  STRUCT
   FC2_RECV_1 : ARRAY  [0 .. 499 ] OF BYTE  := B#16#0;
  END_STRUCT ;
BEGIN
   FC2_RECV_1[0] := B#16#0;
   FC2_RECV_1[1] := B#16#0;
   FC2_RECV_1[2] := B#16#0;
   FC2_RECV_1[3] := B#16#0;
   FC2_RECV_1[4] := B#16#0;
   FC2_RECV_1[5] := B#16#0;
   FC2_RECV_1[6] := B#16#0;
   FC2_RECV_1[7] := B#16#0;
   FC2_RECV_1[8] := B#16#0;
   FC2_RECV_1[9] := B#16#0;
   FC2_RECV_1[10] := B#16#0;
   FC2_RECV_1[11] := B#16#0;
   FC2_RECV_1[12] := B#16#0;
   FC2_RECV_1[13] := B#16#0;
   FC2_RECV_1[14] := B#16#0;
   FC2_RECV_1[15] := B#16#0;
   FC2_RECV_1[16] := B#16#0;
   FC2_RECV_1[17] := B#16#0;
   FC2_RECV_1[18] := B#16#0;
   FC2_RECV_1[19] := B#16#0;
   FC2_RECV_1[20] := B#16#0;
   FC2_RECV_1[21] := B#16#0;
   FC2_RECV_1[22] := B#16#0;
   FC2_RECV_1[23] := B#16#0;
   FC2_RECV_1[24] := B#16#0;
   FC2_RECV_1[25] := B#16#0;
   FC2_RECV_1[26] := B#16#0;
   FC2_RECV_1[27] := B#16#0;
   FC2_RECV_1[28] := B#16#0;
   FC2_RECV_1[29] := B#16#0;
   FC2_RECV_1[30] := B#16#0;
   FC2_RECV_1[31] := B#16#0;
   FC2_RECV_1[32] := B#16#0;
   FC2_RECV_1[33] := B#16#0;
   FC2_RECV_1[34] := B#16#0;
   FC2_RECV_1[35] := B#16#0;
   FC2_RECV_1[36] := B#16#0;
   FC2_RECV_1[37] := B#16#0;
   FC2_RECV_1[38] := B#16#0;
   FC2_RECV_1[39] := B#16#0;
   FC2_RECV_1[40] := B#16#0;
   FC2_RECV_1[41] := B#16#0;
   FC2_RECV_1[42] := B#16#0;
   FC2_RECV_1[43] := B#16#0;
   FC2_RECV_1[44] := B#16#0;
   FC2_RECV_1[45] := B#16#0;
   FC2_RECV_1[46] := B#16#0;
   FC2_RECV_1[47] := B#16#0;
   FC2_RECV_1[48] := B#16#0;
   FC2_RECV_1[49] := B#16#0;
   FC2_RECV_1[50] := B#16#0;
   FC2_RECV_1[51] := B#16#0;
   FC2_RECV_1[52] := B#16#0;
   FC2_RECV_1[53] := B#16#0;
   FC2_RECV_1[54] := B#16#0;
   FC2_RECV_1[55] := B#16#0;
   FC2_RECV_1[56] := B#16#0;
   FC2_RECV_1[57] := B#16#0;
   FC2_RECV_1[58] := B#16#0;
   FC2_RECV_1[59] := B#16#0;
   FC2_RECV_1[60] := B#16#0;
   FC2_RECV_1[61] := B#16#0;
   FC2_RECV_1[62] := B#16#0;
   FC2_RECV_1[63] := B#16#0;
   FC2_RECV_1[64] := B#16#0;
   FC2_RECV_1[65] := B#16#0;
   FC2_RECV_1[66] := B#16#0;
   FC2_RECV_1[67] := B#16#0;
   FC2_RECV_1[68] := B#16#0;
   FC2_RECV_1[69] := B#16#0;
   FC2_RECV_1[70] := B#16#0;
   FC2_RECV_1[71] := B#16#0;
   FC2_RECV_1[72] := B#16#0;
   FC2_RECV_1[73] := B#16#0;
   FC2_RECV_1[74] := B#16#0;
   FC2_RECV_1[75] := B#16#0;
   FC2_RECV_1[76] := B#16#0;
   FC2_RECV_1[77] := B#16#0;
   FC2_RECV_1[78] := B#16#0;
   FC2_RECV_1[79] := B#16#0;
   FC2_RECV_1[80] := B#16#0;
   FC2_RECV_1[81] := B#16#0;
   FC2_RECV_1[82] := B#16#0;
   FC2_RECV_1[83] := B#16#0;
   FC2_RECV_1[84] := B#16#0;
   FC2_RECV_1[85] := B#16#0;
   FC2_RECV_1[86] := B#16#0;
   FC2_RECV_1[87] := B#16#0;
   FC2_RECV_1[88] := B#16#0;
   FC2_RECV_1[89] := B#16#0;
   FC2_RECV_1[90] := B#16#0;
   FC2_RECV_1[91] := B#16#0;
   FC2_RECV_1[92] := B#16#0;
   FC2_RECV_1[93] := B#16#0;
   FC2_RECV_1[94] := B#16#0;
   FC2_RECV_1[95] := B#16#0;
   FC2_RECV_1[96] := B#16#0;
   FC2_RECV_1[97] := B#16#0;
   FC2_RECV_1[98] := B#16#0;
   FC2_RECV_1[99] := B#16#0;
   FC2_RECV_1[100] := B#16#0;
   FC2_RECV_1[101] := B#16#0;
   FC2_RECV_1[102] := B#16#0;
   FC2_RECV_1[103] := B#16#0;
   FC2_RECV_1[104] := B#16#0;
   FC2_RECV_1[105] := B#16#0;
   FC2_RECV_1[106] := B#16#0;
   FC2_RECV_1[107] := B#16#0;
   FC2_RECV_1[108] := B#16#0;
   FC2_RECV_1[109] := B#16#0;
   FC2_RECV_1[110] := B#16#0;
   FC2_RECV_1[111] := B#16#0;
   FC2_RECV_1[112] := B#16#0;
   FC2_RECV_1[113] := B#16#0;
   FC2_RECV_1[114] := B#16#0;
   FC2_RECV_1[115] := B#16#0;
   FC2_RECV_1[116] := B#16#0;
   FC2_RECV_1[117] := B#16#0;
   FC2_RECV_1[118] := B#16#0;
   FC2_RECV_1[119] := B#16#0;
   FC2_RECV_1[120] := B#16#0;
   FC2_RECV_1[121] := B#16#0;
   FC2_RECV_1[122] := B#16#0;
   FC2_RECV_1[123] := B#16#0;
   FC2_RECV_1[124] := B#16#0;
   FC2_RECV_1[125] := B#16#0;
   FC2_RECV_1[126] := B#16#0;
   FC2_RECV_1[127] := B#16#0;
   FC2_RECV_1[128] := B#16#0;
   FC2_RECV_1[129] := B#16#0;
   FC2_RECV_1[130] := B#16#0;
   FC2_RECV_1[131] := B#16#0;
   FC2_RECV_1[132] := B#16#0;
   FC2_RECV_1[133] := B#16#0;
   FC2_RECV_1[134] := B#16#0;
   FC2_RECV_1[135] := B#16#0;
   FC2_RECV_1[136] := B#16#0;
   FC2_RECV_1[137] := B#16#0;
   FC2_RECV_1[138] := B#16#0;
   FC2_RECV_1[139] := B#16#0;
   FC2_RECV_1[140] := B#16#0;
   FC2_RECV_1[141] := B#16#0;
   FC2_RECV_1[142] := B#16#0;
   FC2_RECV_1[143] := B#16#0;
   FC2_RECV_1[144] := B#16#0;
   FC2_RECV_1[145] := B#16#0;
   FC2_RECV_1[146] := B#16#0;
   FC2_RECV_1[147] := B#16#0;
   FC2_RECV_1[148] := B#16#0;
   FC2_RECV_1[149] := B#16#0;
   FC2_RECV_1[150] := B#16#0;
   FC2_RECV_1[151] := B#16#0;
   FC2_RECV_1[152] := B#16#0;
   FC2_RECV_1[153] := B#16#0;
   FC2_RECV_1[154] := B#16#0;
   FC2_RECV_1[155] := B#16#0;
   FC2_RECV_1[156] := B#16#0;
   FC2_RECV_1[157] := B#16#0;
   FC2_RECV_1[158] := B#16#0;
   FC2_RECV_1[159] := B#16#0;
   FC2_RECV_1[160] := B#16#0;
   FC2_RECV_1[161] := B#16#0;
   FC2_RECV_1[162] := B#16#0;
   FC2_RECV_1[163] := B#16#0;
   FC2_RECV_1[164] := B#16#0;
   FC2_RECV_1[165] := B#16#0;
   FC2_RECV_1[166] := B#16#0;
   FC2_RECV_1[167] := B#16#0;
   FC2_RECV_1[168] := B#16#0;
   FC2_RECV_1[169] := B#16#0;
   FC2_RECV_1[170] := B#16#0;
   FC2_RECV_1[171] := B#16#0;
   FC2_RECV_1[172] := B#16#0;
   FC2_RECV_1[173] := B#16#0;
   FC2_RECV_1[174] := B#16#0;
   FC2_RECV_1[175] := B#16#0;
   FC2_RECV_1[176] := B#16#0;
   FC2_RECV_1[177] := B#16#0;
   FC2_RECV_1[178] := B#16#0;
   FC2_RECV_1[179] := B#16#0;
   FC2_RECV_1[180] := B#16#0;
   FC2_RECV_1[181] := B#16#0;
   FC2_RECV_1[182] := B#16#0;
   FC2_RECV_1[183] := B#16#0;
   FC2_RECV_1[184] := B#16#0;
   FC2_RECV_1[185] := B#16#0;
   FC2_RECV_1[186] := B#16#0;
   FC2_RECV_1[187] := B#16#0;
   FC2_RECV_1[188] := B#16#0;
   FC2_RECV_1[189] := B#16#0;
   FC2_RECV_1[190] := B#16#0;
   FC2_RECV_1[191] := B#16#0;
   FC2_RECV_1[192] := B#16#0;
   FC2_RECV_1[193] := B#16#0;
   FC2_RECV_1[194] := B#16#0;
   FC2_RECV_1[195] := B#16#0;
   FC2_RECV_1[196] := B#16#0;
   FC2_RECV_1[197] := B#16#0;
   FC2_RECV_1[198] := B#16#0;
   FC2_RECV_1[199] := B#16#0;
   FC2_RECV_1[200] := B#16#0;
   FC2_RECV_1[201] := B#16#0;
   FC2_RECV_1[202] := B#16#0;
   FC2_RECV_1[203] := B#16#0;
   FC2_RECV_1[204] := B#16#0;
   FC2_RECV_1[205] := B#16#0;
   FC2_RECV_1[206] := B#16#0;
   FC2_RECV_1[207] := B#16#0;
   FC2_RECV_1[208] := B#16#0;
   FC2_RECV_1[209] := B#16#0;
   FC2_RECV_1[210] := B#16#0;
   FC2_RECV_1[211] := B#16#0;
   FC2_RECV_1[212] := B#16#0;
   FC2_RECV_1[213] := B#16#0;
   FC2_RECV_1[214] := B#16#0;
   FC2_RECV_1[215] := B#16#0;
   FC2_RECV_1[216] := B#16#0;
   FC2_RECV_1[217] := B#16#0;
   FC2_RECV_1[218] := B#16#0;
   FC2_RECV_1[219] := B#16#0;
   FC2_RECV_1[220] := B#16#0;
   FC2_RECV_1[221] := B#16#0;
   FC2_RECV_1[222] := B#16#0;
   FC2_RECV_1[223] := B#16#0;
   FC2_RECV_1[224] := B#16#0;
   FC2_RECV_1[225] := B#16#0;
   FC2_RECV_1[226] := B#16#0;
   FC2_RECV_1[227] := B#16#0;
   FC2_RECV_1[228] := B#16#0;
   FC2_RECV_1[229] := B#16#0;
   FC2_RECV_1[230] := B#16#0;
   FC2_RECV_1[231] := B#16#0;
   FC2_RECV_1[232] := B#16#0;
   FC2_RECV_1[233] := B#16#0;
   FC2_RECV_1[234] := B#16#0;
   FC2_RECV_1[235] := B#16#0;
   FC2_RECV_1[236] := B#16#0;
   FC2_RECV_1[237] := B#16#0;
   FC2_RECV_1[238] := B#16#0;
   FC2_RECV_1[239] := B#16#0;
   FC2_RECV_1[240] := B#16#0;
   FC2_RECV_1[241] := B#16#0;
   FC2_RECV_1[242] := B#16#0;
   FC2_RECV_1[243] := B#16#0;
   FC2_RECV_1[244] := B#16#0;
   FC2_RECV_1[245] := B#16#0;
   FC2_RECV_1[246] := B#16#0;
   FC2_RECV_1[247] := B#16#0;
   FC2_RECV_1[248] := B#16#0;
   FC2_RECV_1[249] := B#16#0;
   FC2_RECV_1[250] := B#16#0;
   FC2_RECV_1[251] := B#16#0;
   FC2_RECV_1[252] := B#16#0;
   FC2_RECV_1[253] := B#16#0;
   FC2_RECV_1[254] := B#16#0;
   FC2_RECV_1[255] := B#16#0;
   FC2_RECV_1[256] := B#16#0;
   FC2_RECV_1[257] := B#16#0;
   FC2_RECV_1[258] := B#16#0;
   FC2_RECV_1[259] := B#16#0;
   FC2_RECV_1[260] := B#16#0;
   FC2_RECV_1[261] := B#16#0;
   FC2_RECV_1[262] := B#16#0;
   FC2_RECV_1[263] := B#16#0;
   FC2_RECV_1[264] := B#16#0;
   FC2_RECV_1[265] := B#16#0;
   FC2_RECV_1[266] := B#16#0;
   FC2_RECV_1[267] := B#16#0;
   FC2_RECV_1[268] := B#16#0;
   FC2_RECV_1[269] := B#16#0;
   FC2_RECV_1[270] := B#16#0;
   FC2_RECV_1[271] := B#16#0;
   FC2_RECV_1[272] := B#16#0;
   FC2_RECV_1[273] := B#16#0;
   FC2_RECV_1[274] := B#16#0;
   FC2_RECV_1[275] := B#16#0;
   FC2_RECV_1[276] := B#16#0;
   FC2_RECV_1[277] := B#16#0;
   FC2_RECV_1[278] := B#16#0;
   FC2_RECV_1[279] := B#16#0;
   FC2_RECV_1[280] := B#16#0;
   FC2_RECV_1[281] := B#16#0;
   FC2_RECV_1[282] := B#16#0;
   FC2_RECV_1[283] := B#16#0;
   FC2_RECV_1[284] := B#16#0;
   FC2_RECV_1[285] := B#16#0;
   FC2_RECV_1[286] := B#16#0;
   FC2_RECV_1[287] := B#16#0;
   FC2_RECV_1[288] := B#16#0;
   FC2_RECV_1[289] := B#16#0;
   FC2_RECV_1[290] := B#16#0;
   FC2_RECV_1[291] := B#16#0;
   FC2_RECV_1[292] := B#16#0;
   FC2_RECV_1[293] := B#16#0;
   FC2_RECV_1[294] := B#16#0;
   FC2_RECV_1[295] := B#16#0;
   FC2_RECV_1[296] := B#16#0;
   FC2_RECV_1[297] := B#16#0;
   FC2_RECV_1[298] := B#16#0;
   FC2_RECV_1[299] := B#16#0;
   FC2_RECV_1[300] := B#16#0;
   FC2_RECV_1[301] := B#16#0;
   FC2_RECV_1[302] := B#16#0;
   FC2_RECV_1[303] := B#16#0;
   FC2_RECV_1[304] := B#16#0;
   FC2_RECV_1[305] := B#16#0;
   FC2_RECV_1[306] := B#16#0;
   FC2_RECV_1[307] := B#16#0;
   FC2_RECV_1[308] := B#16#0;
   FC2_RECV_1[309] := B#16#0;
   FC2_RECV_1[310] := B#16#0;
   FC2_RECV_1[311] := B#16#0;
   FC2_RECV_1[312] := B#16#0;
   FC2_RECV_1[313] := B#16#0;
   FC2_RECV_1[314] := B#16#0;
   FC2_RECV_1[315] := B#16#0;
   FC2_RECV_1[316] := B#16#0;
   FC2_RECV_1[317] := B#16#0;
   FC2_RECV_1[318] := B#16#0;
   FC2_RECV_1[319] := B#16#0;
   FC2_RECV_1[320] := B#16#0;
   FC2_RECV_1[321] := B#16#0;
   FC2_RECV_1[322] := B#16#0;
   FC2_RECV_1[323] := B#16#0;
   FC2_RECV_1[324] := B#16#0;
   FC2_RECV_1[325] := B#16#0;
   FC2_RECV_1[326] := B#16#0;
   FC2_RECV_1[327] := B#16#0;
   FC2_RECV_1[328] := B#16#0;
   FC2_RECV_1[329] := B#16#0;
   FC2_RECV_1[330] := B#16#0;
   FC2_RECV_1[331] := B#16#0;
   FC2_RECV_1[332] := B#16#0;
   FC2_RECV_1[333] := B#16#0;
   FC2_RECV_1[334] := B#16#0;
   FC2_RECV_1[335] := B#16#0;
   FC2_RECV_1[336] := B#16#0;
   FC2_RECV_1[337] := B#16#0;
   FC2_RECV_1[338] := B#16#0;
   FC2_RECV_1[339] := B#16#0;
   FC2_RECV_1[340] := B#16#0;
   FC2_RECV_1[341] := B#16#0;
   FC2_RECV_1[342] := B#16#0;
   FC2_RECV_1[343] := B#16#0;
   FC2_RECV_1[344] := B#16#0;
   FC2_RECV_1[345] := B#16#0;
   FC2_RECV_1[346] := B#16#0;
   FC2_RECV_1[347] := B#16#0;
   FC2_RECV_1[348] := B#16#0;
   FC2_RECV_1[349] := B#16#0;
   FC2_RECV_1[350] := B#16#0;
   FC2_RECV_1[351] := B#16#0;
   FC2_RECV_1[352] := B#16#0;
   FC2_RECV_1[353] := B#16#0;
   FC2_RECV_1[354] := B#16#0;
   FC2_RECV_1[355] := B#16#0;
   FC2_RECV_1[356] := B#16#0;
   FC2_RECV_1[357] := B#16#0;
   FC2_RECV_1[358] := B#16#0;
   FC2_RECV_1[359] := B#16#0;
   FC2_RECV_1[360] := B#16#0;
   FC2_RECV_1[361] := B#16#0;
   FC2_RECV_1[362] := B#16#0;
   FC2_RECV_1[363] := B#16#0;
   FC2_RECV_1[364] := B#16#0;
   FC2_RECV_1[365] := B#16#0;
   FC2_RECV_1[366] := B#16#0;
   FC2_RECV_1[367] := B#16#0;
   FC2_RECV_1[368] := B#16#0;
   FC2_RECV_1[369] := B#16#0;
   FC2_RECV_1[370] := B#16#0;
   FC2_RECV_1[371] := B#16#0;
   FC2_RECV_1[372] := B#16#0;
   FC2_RECV_1[373] := B#16#0;
   FC2_RECV_1[374] := B#16#0;
   FC2_RECV_1[375] := B#16#0;
   FC2_RECV_1[376] := B#16#0;
   FC2_RECV_1[377] := B#16#0;
   FC2_RECV_1[378] := B#16#0;
   FC2_RECV_1[379] := B#16#0;
   FC2_RECV_1[380] := B#16#0;
   FC2_RECV_1[381] := B#16#0;
   FC2_RECV_1[382] := B#16#0;
   FC2_RECV_1[383] := B#16#0;
   FC2_RECV_1[384] := B#16#0;
   FC2_RECV_1[385] := B#16#0;
   FC2_RECV_1[386] := B#16#0;
   FC2_RECV_1[387] := B#16#0;
   FC2_RECV_1[388] := B#16#0;
   FC2_RECV_1[389] := B#16#0;
   FC2_RECV_1[390] := B#16#0;
   FC2_RECV_1[391] := B#16#0;
   FC2_RECV_1[392] := B#16#0;
   FC2_RECV_1[393] := B#16#0;
   FC2_RECV_1[394] := B#16#0;
   FC2_RECV_1[395] := B#16#0;
   FC2_RECV_1[396] := B#16#0;
   FC2_RECV_1[397] := B#16#0;
   FC2_RECV_1[398] := B#16#0;
   FC2_RECV_1[399] := B#16#0;
   FC2_RECV_1[400] := B#16#0;
   FC2_RECV_1[401] := B#16#0;
   FC2_RECV_1[402] := B#16#0;
   FC2_RECV_1[403] := B#16#0;
   FC2_RECV_1[404] := B#16#0;
   FC2_RECV_1[405] := B#16#0;
   FC2_RECV_1[406] := B#16#0;
   FC2_RECV_1[407] := B#16#0;
   FC2_RECV_1[408] := B#16#0;
   FC2_RECV_1[409] := B#16#0;
   FC2_RECV_1[410] := B#16#0;
   FC2_RECV_1[411] := B#16#0;
   FC2_RECV_1[412] := B#16#0;
   FC2_RECV_1[413] := B#16#0;
   FC2_RECV_1[414] := B#16#0;
   FC2_RECV_1[415] := B#16#0;
   FC2_RECV_1[416] := B#16#0;
   FC2_RECV_1[417] := B#16#0;
   FC2_RECV_1[418] := B#16#0;
   FC2_RECV_1[419] := B#16#0;
   FC2_RECV_1[420] := B#16#0;
   FC2_RECV_1[421] := B#16#0;
   FC2_RECV_1[422] := B#16#0;
   FC2_RECV_1[423] := B#16#0;
   FC2_RECV_1[424] := B#16#0;
   FC2_RECV_1[425] := B#16#0;
   FC2_RECV_1[426] := B#16#0;
   FC2_RECV_1[427] := B#16#0;
   FC2_RECV_1[428] := B#16#0;
   FC2_RECV_1[429] := B#16#0;
   FC2_RECV_1[430] := B#16#0;
   FC2_RECV_1[431] := B#16#0;
   FC2_RECV_1[432] := B#16#0;
   FC2_RECV_1[433] := B#16#0;
   FC2_RECV_1[434] := B#16#0;
   FC2_RECV_1[435] := B#16#0;
   FC2_RECV_1[436] := B#16#0;
   FC2_RECV_1[437] := B#16#0;
   FC2_RECV_1[438] := B#16#0;
   FC2_RECV_1[439] := B#16#0;
   FC2_RECV_1[440] := B#16#0;
   FC2_RECV_1[441] := B#16#0;
   FC2_RECV_1[442] := B#16#0;
   FC2_RECV_1[443] := B#16#0;
   FC2_RECV_1[444] := B#16#0;
   FC2_RECV_1[445] := B#16#0;
   FC2_RECV_1[446] := B#16#0;
   FC2_RECV_1[447] := B#16#0;
   FC2_RECV_1[448] := B#16#0;
   FC2_RECV_1[449] := B#16#0;
   FC2_RECV_1[450] := B#16#0;
   FC2_RECV_1[451] := B#16#0;
   FC2_RECV_1[452] := B#16#0;
   FC2_RECV_1[453] := B#16#0;
   FC2_RECV_1[454] := B#16#0;
   FC2_RECV_1[455] := B#16#0;
   FC2_RECV_1[456] := B#16#0;
   FC2_RECV_1[457] := B#16#0;
   FC2_RECV_1[458] := B#16#0;
   FC2_RECV_1[459] := B#16#0;
   FC2_RECV_1[460] := B#16#0;
   FC2_RECV_1[461] := B#16#0;
   FC2_RECV_1[462] := B#16#0;
   FC2_RECV_1[463] := B#16#0;
   FC2_RECV_1[464] := B#16#0;
   FC2_RECV_1[465] := B#16#0;
   FC2_RECV_1[466] := B#16#0;
   FC2_RECV_1[467] := B#16#0;
   FC2_RECV_1[468] := B#16#0;
   FC2_RECV_1[469] := B#16#0;
   FC2_RECV_1[470] := B#16#0;
   FC2_RECV_1[471] := B#16#0;
   FC2_RECV_1[472] := B#16#0;
   FC2_RECV_1[473] := B#16#0;
   FC2_RECV_1[474] := B#16#0;
   FC2_RECV_1[475] := B#16#0;
   FC2_RECV_1[476] := B#16#0;
   FC2_RECV_1[477] := B#16#0;
   FC2_RECV_1[478] := B#16#0;
   FC2_RECV_1[479] := B#16#0;
   FC2_RECV_1[480] := B#16#0;
   FC2_RECV_1[481] := B#16#0;
   FC2_RECV_1[482] := B#16#0;
   FC2_RECV_1[483] := B#16#0;
   FC2_RECV_1[484] := B#16#0;
   FC2_RECV_1[485] := B#16#0;
   FC2_RECV_1[486] := B#16#0;
   FC2_RECV_1[487] := B#16#0;
   FC2_RECV_1[488] := B#16#0;
   FC2_RECV_1[489] := B#16#0;
   FC2_RECV_1[490] := B#16#0;
   FC2_RECV_1[491] := B#16#0;
   FC2_RECV_1[492] := B#16#0;
   FC2_RECV_1[493] := B#16#0;
   FC2_RECV_1[494] := B#16#0;
   FC2_RECV_1[495] := B#16#0;
   FC2_RECV_1[496] := B#16#0;
   FC2_RECV_1[497] := B#16#0;
   FC2_RECV_1[498] := B#16#0;
   FC2_RECV_1[499] := B#16#0;
END_DATA_BLOCK

DATA_BLOCK DB 98
VERSION : 0.1


  STRUCT
   STAT0 : ARRAY  [0 .. 25 ] OF DWORD ;
  END_STRUCT ;
BEGIN
   STAT0[0] := DW#16#0;
   STAT0[1] := DW#16#0;
   STAT0[2] := DW#16#0;
   STAT0[3] := DW#16#0;
   STAT0[4] := DW#16#0;
   STAT0[5] := DW#16#0;
   STAT0[6] := DW#16#0;
   STAT0[7] := DW#16#0;
   STAT0[8] := DW#16#0;
   STAT0[9] := DW#16#0;
   STAT0[10] := DW#16#10000;
   STAT0[11] := DW#16#0;
   STAT0[12] := DW#16#0;
   STAT0[13] := DW#16#0;
   STAT0[14] := DW#16#0;
   STAT0[15] := DW#16#0;
   STAT0[16] := DW#16#0;
   STAT0[17] := DW#16#0;
   STAT0[18] := DW#16#0;
   STAT0[19] := DW#16#0;
   STAT0[20] := DW#16#0;
   STAT0[21] := DW#16#0;
   STAT0[22] := DW#16#0;
   STAT0[23] := DW#16#0;
   STAT0[24] := DW#16#0;
   STAT0[25] := DW#16#0;
END_DATA_BLOCK

DATA_BLOCK DB 99
VERSION : 0.1


  STRUCT
   STAT0 : WORD ;
   STAT1 : WORD ;
   STAT2 : WORD ;
   STAT3 : WORD ;
   STAT4 : WORD ;
   STAT5 : WORD ;
   STAT6 : WORD ;
   STAT7 : WORD ;
   STAT8 : WORD ;
   STAT9 : WORD ;
   STAT10 : WORD ;
   STAT11 : WORD ;
   STAT12 : WORD ;
   STAT13 : WORD ;
   STAT14 : WORD ;
   STAT15 : WORD ;
   STAT16 : WORD ;
   STAT17 : WORD ;
   STAT18 : WORD ;
   STAT19 : WORD ;
   STAT20 : WORD ;
   STAT21 : WORD ;
   STAT22 : WORD ;
   STAT23 : WORD ;
   STAT24 : WORD ;
   STAT25 : WORD ;
   STAT26 : WORD ;
   STAT27 : WORD ;
   STAT28 : WORD ;
   STAT29 : WORD ;
   STAT30 : WORD ;
   STAT31 : WORD ;
   STAT32 : WORD ;
   STAT33 : WORD ;
   STAT34 : WORD ;
   STAT35 : WORD ;
   STAT36 : WORD ;
   STAT37 : WORD ;
   STAT38 : WORD ;
   STAT39 : WORD ;
   STAT40 : WORD ;
   STAT41 : WORD ;
   STAT42 : WORD ;
   STAT43 : WORD ;
   STAT44 : WORD ;
   STAT45 : WORD ;
   STAT46 : WORD ;
   STAT47 : WORD ;
   STAT48 : WORD ;
   STAT49 : WORD ;
   STAT50 : WORD ;
   STAT51 : WORD ;
   STAT52 : WORD ;
   STAT53 : WORD ;
   STAT54 : WORD ;
   STAT55 : WORD ;
   STAT56 : WORD ;
   STAT57 : WORD ;
   STAT58 : WORD ;
   STAT59 : WORD ;
   STAT60 : WORD ;
   STAT61 : WORD ;
   STAT62 : WORD ;
   STAT63 : WORD ;
  END_STRUCT ;
BEGIN
   STAT0 := W#16#4101;
   STAT1 := W#16#9000;
   STAT2 := W#16#800;
   STAT3 := W#16#0;
   STAT4 := W#16#4102;
   STAT5 := W#16#9000;
   STAT6 := W#16#800;
   STAT7 := W#16#0;
   STAT8 := W#16#4201;
   STAT9 := W#16#5000;
   STAT10 := W#16#800;
   STAT11 := W#16#0;
   STAT12 := W#16#4102;
   STAT13 := W#16#9000;
   STAT14 := W#16#800;
   STAT15 := W#16#0;
   STAT16 := W#16#4101;
   STAT17 := W#16#9000;
   STAT18 := W#16#800;
   STAT19 := W#16#0;
   STAT20 := W#16#4101;
   STAT21 := W#16#9000;
   STAT22 := W#16#800;
   STAT23 := W#16#0;
   STAT24 := W#16#0;
   STAT25 := W#16#0;
   STAT26 := W#16#0;
   STAT27 := W#16#0;
   STAT28 := W#16#0;
   STAT29 := W#16#0;
   STAT30 := W#16#0;
   STAT31 := W#16#0;
   STAT32 := W#16#0;
   STAT33 := W#16#0;
   STAT34 := W#16#0;
   STAT35 := W#16#0;
   STAT36 := W#16#0;
   STAT37 := W#16#0;
   STAT38 := W#16#0;
   STAT39 := W#16#0;
   STAT40 := W#16#0;
   STAT41 := W#16#0;
   STAT42 := W#16#0;
   STAT43 := W#16#0;
   STAT44 := W#16#0;
   STAT45 := W#16#4102;
   STAT46 := W#16#9000;
   STAT47 := W#16#4201;
   STAT48 := W#16#5000;
   STAT49 := W#16#4102;
   STAT50 := W#16#9000;
   STAT51 := W#16#4201;
   STAT52 := W#16#5000;
   STAT53 := W#16#4101;
   STAT54 := W#16#9000;
   STAT55 := W#16#800;
   STAT56 := W#16#0;
   STAT57 := W#16#0;
   STAT58 := W#16#0;
   STAT59 := W#16#0;
   STAT60 := W#16#0;
   STAT61 := W#16#0;
   STAT62 := W#16#0;
   STAT63 := W#16#0;
END_DATA_BLOCK

DATA_BLOCK DB 100
VERSION : 0.1


  STRUCT
   STAT0 : WORD ;
   STAT1 : WORD ;
   STAT2 : WORD ;
   STAT3 : WORD ;
   STAT4 : WORD ;
   STAT5 : WORD ;
   STAT6 : WORD ;
   STAT7 : WORD ;
   STAT8 : WORD ;
   STAT9 : WORD ;
   STAT10 : WORD ;
   STAT11 : WORD ;
   STAT12 : WORD ;
   STAT13 : WORD ;
   STAT14 : WORD ;
   STAT15 : WORD ;
   STAT16 : WORD ;
   STAT17 : WORD ;
   STAT18 : WORD ;
   STAT19 : WORD ;
   STAT20 : WORD ;
   STAT21 : WORD ;
   STAT22 : WORD ;
   STAT23 : WORD ;
   STAT24 : WORD ;
   STAT25 : WORD ;
   STAT26 : WORD ;
   STAT27 : WORD ;
   STAT28 : WORD ;
   STAT29 : WORD ;
   STAT30 : WORD ;
   STAT31 : WORD ;
   STAT32 : WORD ;
   STAT33 : WORD ;
   STAT34 : WORD ;
   STAT35 : WORD ;
   STAT36 : WORD ;
   STAT37 : WORD ;
   STAT38 : WORD ;
   STAT39 : WORD ;
   STAT40 : WORD ;
   STAT41 : WORD ;
   STAT42 : WORD ;
   STAT43 : WORD ;
   STAT44 : WORD ;
   STAT45 : WORD ;
   STAT46 : WORD ;
   STAT47 : WORD ;
   STAT48 : WORD ;
   STAT49 : WORD ;
   STAT50 : WORD ;
   STAT51 : WORD ;
   STAT52 : WORD ;
   STAT53 : WORD ;
   STAT54 : WORD ;
   STAT55 : WORD ;
   STAT56 : WORD ;
   STAT57 : WORD ;
   STAT58 : WORD ;
   STAT59 : WORD ;
   STAT60 : WORD ;
   STAT61 : WORD ;
   STAT62 : WORD ;
   STAT63 : WORD ;
   STAT64 : WORD ;
   STAT65 : WORD ;
   STAT66 : WORD ;
   STAT67 : WORD ;
   STAT68 : WORD ;
   STAT69 : WORD ;
   STAT70 : WORD ;
   STAT71 : WORD ;
   STAT72 : WORD ;
   STAT73 : WORD ;
   STAT74 : WORD ;
   STAT75 : WORD ;
   STAT76 : WORD ;
   STAT77 : WORD ;
   STAT78 : WORD ;
   STAT79 : WORD ;
  END_STRUCT ;
BEGIN
   STAT0 := W#16#0;
   STAT1 := W#16#0;
   STAT2 := W#16#0;
   STAT3 := W#16#0;
   STAT4 := W#16#0;
   STAT5 := W#16#0;
   STAT6 := W#16#0;
   STAT7 := W#16#0;
   STAT8 := W#16#4201;
   STAT9 := W#16#5000;
   STAT10 := W#16#800;
   STAT11 := W#16#0;
   STAT12 := W#16#4102;
   STAT13 := W#16#9000;
   STAT14 := W#16#800;
   STAT15 := W#16#0;
   STAT16 := W#16#4101;
   STAT17 := W#16#9000;
   STAT18 := W#16#800;
   STAT19 := W#16#0;
   STAT20 := W#16#4201;
   STAT21 := W#16#5000;
   STAT22 := W#16#800;
   STAT23 := W#16#0;
   STAT24 := W#16#4102;
   STAT25 := W#16#9000;
   STAT26 := W#16#800;
   STAT27 := W#16#0;
   STAT28 := W#16#4101;
   STAT29 := W#16#9000;
   STAT30 := W#16#800;
   STAT31 := W#16#0;
   STAT32 := W#16#4102;
   STAT33 := W#16#A000;
   STAT34 := W#16#1000;
   STAT35 := W#16#0;
   STAT36 := W#16#4201;
   STAT37 := W#16#5000;
   STAT38 := W#16#800;
   STAT39 := W#16#0;
   STAT40 := W#16#4101;
   STAT41 := W#16#9000;
   STAT42 := W#16#800;
   STAT43 := W#16#0;
   STAT44 := W#16#0;
   STAT45 := W#16#0;
   STAT46 := W#16#0;
   STAT47 := W#16#0;
   STAT48 := W#16#0;
   STAT49 := W#16#0;
   STAT50 := W#16#0;
   STAT51 := W#16#0;
   STAT52 := W#16#0;
   STAT53 := W#16#0;
   STAT54 := W#16#0;
   STAT55 := W#16#0;
   STAT56 := W#16#0;
   STAT57 := W#16#0;
   STAT58 := W#16#0;
   STAT59 := W#16#0;
   STAT60 := W#16#0;
   STAT61 := W#16#0;
   STAT62 := W#16#0;
   STAT63 := W#16#0;
   STAT64 := W#16#0;
   STAT65 := W#16#0;
   STAT66 := W#16#0;
   STAT67 := W#16#0;
   STAT68 := W#16#0;
   STAT69 := W#16#0;
   STAT70 := W#16#0;
   STAT71 := W#16#0;
   STAT72 := W#16#0;
   STAT73 := W#16#0;
   STAT74 := W#16#0;
   STAT75 := W#16#0;
   STAT76 := W#16#0;
   STAT77 := W#16#0;
   STAT78 := W#16#0;
   STAT79 := W#16#0;
END_DATA_BLOCK

DATA_BLOCK DB 101
VERSION : 0.1


  STRUCT
   STAT0 : ARRAY  [0 .. 100 ] OF BYTE  := B#16#0;
  END_STRUCT ;
BEGIN
   STAT0[0] := B#16#0;
   STAT0[1] := B#16#0;
   STAT0[2] := B#16#0;
   STAT0[3] := B#16#0;
   STAT0[4] := B#16#0;
   STAT0[5] := B#16#0;
   STAT0[6] := B#16#0;
   STAT0[7] := B#16#0;
   STAT0[8] := B#16#0;
   STAT0[9] := B#16#0;
   STAT0[10] := B#16#0;
   STAT0[11] := B#16#0;
   STAT0[12] := B#16#0;
   STAT0[13] := B#16#0;
   STAT0[14] := B#16#0;
   STAT0[15] := B#16#0;
   STAT0[16] := B#16#0;
   STAT0[17] := B#16#0;
   STAT0[18] := B#16#0;
   STAT0[19] := B#16#0;
   STAT0[20] := B#16#0;
   STAT0[21] := B#16#0;
   STAT0[22] := B#16#0;
   STAT0[23] := B#16#0;
   STAT0[24] := B#16#0;
   STAT0[25] := B#16#0;
   STAT0[26] := B#16#0;
   STAT0[27] := B#16#0;
   STAT0[28] := B#16#0;
   STAT0[29] := B#16#0;
   STAT0[30] := B#16#0;
   STAT0[31] := B#16#0;
   STAT0[32] := B#16#0;
   STAT0[33] := B#16#0;
   STAT0[34] := B#16#0;
   STAT0[35] := B#16#0;
   STAT0[36] := B#16#0;
   STAT0[37] := B#16#0;
   STAT0[38] := B#16#0;
   STAT0[39] := B#16#0;
   STAT0[40] := B#16#0;
   STAT0[41] := B#16#0;
   STAT0[42] := B#16#0;
   STAT0[43] := B#16#0;
   STAT0[44] := B#16#0;
   STAT0[45] := B#16#0;
   STAT0[46] := B#16#0;
   STAT0[47] := B#16#0;
   STAT0[48] := B#16#0;
   STAT0[49] := B#16#0;
   STAT0[50] := B#16#0;
   STAT0[51] := B#16#0;
   STAT0[52] := B#16#0;
   STAT0[53] := B#16#0;
   STAT0[54] := B#16#0;
   STAT0[55] := B#16#0;
   STAT0[56] := B#16#0;
   STAT0[57] := B#16#0;
   STAT0[58] := B#16#0;
   STAT0[59] := B#16#0;
   STAT0[60] := B#16#0;
   STAT0[61] := B#16#0;
   STAT0[62] := B#16#0;
   STAT0[63] := B#16#0;
   STAT0[64] := B#16#0;
   STAT0[65] := B#16#0;
   STAT0[66] := B#16#0;
   STAT0[67] := B#16#0;
   STAT0[68] := B#16#0;
   STAT0[69] := B#16#0;
   STAT0[70] := B#16#0;
   STAT0[71] := B#16#0;
   STAT0[72] := B#16#0;
   STAT0[73] := B#16#0;
   STAT0[74] := B#16#0;
   STAT0[75] := B#16#0;
   STAT0[76] := B#16#0;
   STAT0[77] := B#16#0;
   STAT0[78] := B#16#0;
   STAT0[79] := B#16#0;
   STAT0[80] := B#16#0;
   STAT0[81] := B#16#0;
   STAT0[82] := B#16#0;
   STAT0[83] := B#16#0;
   STAT0[84] := B#16#0;
   STAT0[85] := B#16#0;
   STAT0[86] := B#16#0;
   STAT0[87] := B#16#0;
   STAT0[88] := B#16#0;
   STAT0[89] := B#16#0;
   STAT0[90] := B#16#0;
   STAT0[91] := B#16#0;
   STAT0[92] := B#16#0;
   STAT0[93] := B#16#0;
   STAT0[94] := B#16#0;
   STAT0[95] := B#16#0;
   STAT0[96] := B#16#0;
   STAT0[97] := B#16#0;
   STAT0[98] := B#16#0;
   STAT0[99] := B#16#0;
   STAT0[100] := B#16#0;
END_DATA_BLOCK

DATA_BLOCK DB 160
VERSION : 0.1


  STRUCT
   STAT0 : STRUCT
    STAT1 : INT ;
    STAT2 : INT ;
    STAT3 : INT ;
    STAT4 : INT ;
    STAT5 : WORD ;
    STAT6 : WORD ;
    STAT7 : INT ;
    STAT8 : INT ;
    STAT9 : INT ;
    STAT10 : INT ;
    STAT11 : INT ;
    STAT12 : INT ;
    STAT13 : WORD ;
    STAT14 : WORD ;
    STAT15 : WORD ;
    STAT16 : WORD ;
    STAT17 : WORD ;
    STAT18 : WORD ;
    STAT19 : WORD ;
    STAT20 : WORD ;
    STAT21 : WORD ;
    STAT22 : WORD ;
    STAT23 : WORD ;
    STAT24 : WORD ;
    STAT25 : WORD ;
    STAT26 : WORD ;
    STAT27 : WORD ;
    STAT28 : WORD ;
    STAT29 : WORD ;
    STAT30 : WORD ;
   END_STRUCT ;
   STAT31 : STRUCT
    STAT32 : INT ;
    STAT33 : INT ;
    STAT34 : INT ;
    STAT35 : INT ;
    STAT36 : WORD ;
    STAT37 : WORD ;
    STAT38 : INT ;
    STAT39 : INT ;
    STAT40 : INT ;
    STAT41 : INT ;
    STAT42 : INT ;
    STAT43 : INT ;
    STAT44 : WORD ;
    STAT45 : WORD ;
    STAT46 : WORD ;
    STAT47 : WORD ;
    STAT48 : WORD ;
    STAT49 : WORD ;
    STAT50 : WORD ;
    STAT51 : WORD ;
    STAT52 : WORD ;
    STAT53 : WORD ;
    STAT54 : WORD ;
    STAT55 : WORD ;
    STAT56 : WORD ;
    STAT57 : WORD ;
    STAT58 : WORD ;
    STAT59 : WORD ;
    STAT60 : WORD ;
    STAT61 : WORD ;
   END_STRUCT ;
   STAT62 : STRUCT
    STAT63 : INT ;
    STAT64 : INT ;
    STAT65 : INT ;
    STAT66 : INT ;
    STAT67 : WORD ;
    STAT68 : WORD ;
    STAT69 : INT ;
    STAT70 : INT ;
    STAT71 : INT ;
    STAT72 : INT ;
    STAT73 : INT ;
    STAT74 : INT ;
    STAT75 : WORD ;
    STAT76 : WORD ;
    STAT77 : WORD ;
    STAT78 : WORD ;
    STAT79 : WORD ;
    STAT80 : WORD ;
    STAT81 : WORD ;
    STAT82 : WORD ;
    STAT83 : WORD ;
    STAT84 : WORD ;
    STAT85 : WORD ;
    STAT86 : WORD ;
    STAT87 : WORD ;
    STAT88 : WORD ;
    STAT89 : WORD ;
    STAT90 : WORD ;
    STAT91 : WORD ;
    STAT92 : WORD ;
   END_STRUCT ;
   STAT93 : STRUCT
    STAT94 : INT ;
    STAT95 : INT ;
    STAT96 : INT ;
    STAT97 : INT ;
    STAT98 : WORD ;
    STAT99 : WORD ;
    STAT100 : INT ;
    STAT101 : INT ;
    STAT102 : INT ;
    STAT103 : INT ;
    STAT104 : INT ;
    STAT105 : INT ;
    STAT106 : WORD ;
    STAT107 : WORD ;
    STAT108 : WORD ;
    STAT109 : WORD ;
    STAT110 : WORD ;
    STAT111 : WORD ;
    STAT112 : WORD ;
    STAT113 : WORD ;
    STAT114 : WORD ;
    STAT115 : WORD ;
    STAT116 : WORD ;
    STAT117 : WORD ;
    STAT118 : WORD ;
    STAT119 : WORD ;
    STAT120 : WORD ;
    STAT121 : WORD ;
    STAT122 : WORD ;
    STAT123 : WORD ;
   END_STRUCT ;
   STAT124 : STRUCT
    STAT125 : INT ;
    STAT126 : INT ;
    STAT127 : INT ;
    STAT128 : INT ;
    STAT129 : WORD ;
    STAT130 : WORD ;
    STAT131 : INT ;
    STAT132 : INT ;
    STAT133 : INT ;
    STAT134 : INT ;
    STAT135 : INT ;
    STAT136 : INT ;
    STAT137 : WORD ;
    STAT138 : WORD ;
    STAT139 : WORD ;
    STAT140 : WORD ;
    STAT141 : WORD ;
    STAT142 : WORD ;
    STAT143 : WORD ;
    STAT144 : WORD ;
    STAT145 : WORD ;
    STAT146 : WORD ;
    STAT147 : WORD ;
    STAT148 : WORD ;
    STAT149 : WORD ;
    STAT150 : WORD ;
    STAT151 : WORD ;
    STAT152 : WORD ;
    STAT153 : WORD ;
    STAT154 : WORD ;
   END_STRUCT ;
   STAT155 : STRUCT
    STAT156 : INT ;
    STAT157 : INT ;
    STAT158 : INT ;
    STAT159 : INT ;
    STAT160 : WORD ;
    STAT161 : WORD ;
    STAT162 : INT ;
    STAT163 : INT ;
    STAT164 : INT ;
    STAT165 : INT ;
    STAT166 : INT ;
    STAT167 : INT ;
    STAT168 : WORD ;
    STAT169 : WORD ;
    STAT170 : WORD ;
    STAT171 : WORD ;
    STAT172 : WORD ;
    STAT173 : WORD ;
    STAT174 : WORD ;
    STAT175 : WORD ;
    STAT176 : WORD ;
    STAT177 : WORD ;
    STAT178 : WORD ;
    STAT179 : WORD ;
    STAT180 : WORD ;
    STAT181 : WORD ;
    STAT182 : WORD ;
    STAT183 : WORD ;
    STAT184 : WORD ;
    STAT185 : WORD ;
   END_STRUCT ;
   STAT186 : STRUCT
    STAT187 : INT ;
    STAT188 : INT ;
    STAT189 : INT ;
    STAT190 : INT ;
    STAT191 : WORD ;
    STAT192 : WORD ;
    STAT193 : INT ;
    STAT194 : INT ;
    STAT195 : INT ;
    STAT196 : INT ;
    STAT197 : INT ;
    STAT198 : INT ;
    STAT199 : WORD ;
    STAT200 : WORD ;
    STAT201 : WORD ;
    STAT202 : WORD ;
    STAT203 : WORD ;
    STAT204 : WORD ;
    STAT205 : WORD ;
    STAT206 : WORD ;
    STAT207 : WORD ;
    STAT208 : WORD ;
    STAT209 : WORD ;
    STAT210 : WORD ;
    STAT211 : WORD ;
    STAT212 : WORD ;
    STAT213 : WORD ;
    STAT214 : WORD ;
    STAT215 : WORD ;
    STAT216 : WORD ;
   END_STRUCT ;
   STAT217 : STRUCT
    STAT218 : INT ;
    STAT219 : INT ;
    STAT220 : INT ;
    STAT221 : INT ;
    STAT222 : WORD ;
    STAT223 : WORD ;
    STAT224 : INT ;
    STAT225 : INT ;
    STAT226 : INT ;
    STAT227 : INT ;
    STAT228 : INT ;
    STAT229 : INT ;
    STAT230 : WORD ;
    STAT231 : WORD ;
    STAT232 : WORD ;
    STAT233 : WORD ;
    STAT234 : WORD ;
    STAT235 : WORD ;
    STAT236 : WORD ;
    STAT237 : WORD ;
    STAT238 : WORD ;
    STAT239 : WORD ;
    STAT240 : WORD ;
    STAT241 : WORD ;
    STAT242 : WORD ;
    STAT243 : WORD ;
    STAT244 : WORD ;
    STAT245 : WORD ;
    STAT246 : WORD ;
    STAT247 : WORD ;
   END_STRUCT ;
   STAT248 : STRUCT
    STAT249 : INT ;
    STAT250 : INT ;
    STAT251 : INT ;
    STAT252 : INT ;
    STAT253 : WORD ;
    STAT254 : WORD ;
    STAT255 : INT ;
    STAT256 : INT ;
    STAT257 : INT ;
    STAT258 : INT ;
    STAT259 : INT ;
    STAT260 : INT ;
    STAT261 : WORD ;
    STAT262 : WORD ;
    STAT263 : WORD ;
    STAT264 : WORD ;
    STAT265 : WORD ;
    STAT266 : WORD ;
    STAT267 : WORD ;
    STAT268 : WORD ;
    STAT269 : WORD ;
    STAT270 : WORD ;
    STAT271 : WORD ;
    STAT272 : WORD ;
    STAT273 : WORD ;
    STAT274 : WORD ;
    STAT275 : WORD ;
    STAT276 : WORD ;
    STAT277 : WORD ;
    STAT278 : WORD ;
   END_STRUCT ;
   STAT279 : STRUCT
    STAT280 : INT ;
    STAT281 : INT ;
    STAT282 : INT ;
    STAT283 : INT ;
    STAT284 : WORD ;
    STAT285 : WORD ;
    STAT286 : INT ;
    STAT287 : INT ;
    STAT288 : INT ;
    STAT289 : INT ;
    STAT290 : INT ;
    STAT291 : INT ;
    STAT292 : WORD ;
    STAT293 : WORD ;
    STAT294 : WORD ;
    STAT295 : WORD ;
    STAT296 : WORD ;
    STAT297 : WORD ;
    STAT298 : WORD ;
    STAT299 : WORD ;
    STAT300 : WORD ;
    STAT301 : WORD ;
    STAT302 : WORD ;
    STAT303 : WORD ;
    STAT304 : WORD ;
    STAT305 : WORD ;
    STAT306 : WORD ;
    STAT307 : WORD ;
    STAT308 : WORD ;
    STAT309 : WORD ;
   END_STRUCT ;
   STAT310 : STRUCT
    STAT311 : INT ;
    STAT312 : INT ;
    STAT313 : INT ;
    STAT314 : INT ;
    STAT315 : WORD ;
    STAT316 : WORD ;
    STAT317 : INT ;
    STAT318 : INT ;
    STAT319 : INT ;
    STAT320 : INT ;
    STAT321 : INT ;
    STAT322 : INT ;
    STAT323 : WORD ;
    STAT324 : WORD ;
    STAT325 : WORD ;
    STAT326 : WORD ;
    STAT327 : WORD ;
    STAT328 : WORD ;
    STAT329 : WORD ;
    STAT330 : WORD ;
    STAT331 : WORD ;
    STAT332 : WORD ;
    STAT333 : WORD ;
    STAT334 : WORD ;
    STAT335 : WORD ;
    STAT336 : WORD ;
    STAT337 : WORD ;
    STAT338 : WORD ;
    STAT339 : WORD ;
    STAT340 : WORD ;
   END_STRUCT ;
   STAT341 : STRUCT
    STAT342 : INT ;
    STAT343 : INT ;
    STAT344 : INT ;
    STAT345 : INT ;
    STAT346 : WORD ;
    STAT347 : WORD ;
    STAT348 : INT ;
    STAT349 : INT ;
    STAT350 : INT ;
    STAT351 : INT ;
    STAT352 : INT ;
    STAT353 : INT ;
    STAT354 : WORD ;
    STAT355 : WORD ;
    STAT356 : WORD ;
    STAT357 : WORD ;
    STAT358 : WORD ;
    STAT359 : WORD ;
    STAT360 : WORD ;
    STAT361 : WORD ;
    STAT362 : WORD ;
    STAT363 : WORD ;
    STAT364 : WORD ;
    STAT365 : WORD ;
    STAT366 : WORD ;
    STAT367 : WORD ;
    STAT368 : WORD ;
    STAT369 : WORD ;
    STAT370 : WORD ;
    STAT371 : WORD ;
   END_STRUCT ;
   STAT372 : STRUCT
    STAT373 : INT ;
    STAT374 : INT ;
    STAT375 : INT ;
    STAT376 : INT ;
    STAT377 : WORD ;
    STAT378 : WORD ;
    STAT379 : INT ;
    STAT380 : INT ;
    STAT381 : INT ;
    STAT382 : INT ;
    STAT383 : INT ;
    STAT384 : INT ;
    STAT385 : WORD ;
    STAT386 : WORD ;
    STAT387 : WORD ;
    STAT388 : WORD ;
    STAT389 : WORD ;
    STAT390 : WORD ;
    STAT391 : WORD ;
    STAT392 : WORD ;
    STAT393 : WORD ;
    STAT394 : WORD ;
    STAT395 : WORD ;
    STAT396 : WORD ;
    STAT397 : WORD ;
    STAT398 : WORD ;
    STAT399 : WORD ;
    STAT400 : WORD ;
    STAT401 : WORD ;
    STAT402 : WORD ;
   END_STRUCT ;
   STAT403 : STRUCT
    STAT404 : INT ;
    STAT405 : INT ;
    STAT406 : INT ;
    STAT407 : INT ;
    STAT408 : WORD ;
    STAT409 : WORD ;
    STAT410 : INT ;
    STAT411 : INT ;
    STAT412 : INT ;
    STAT413 : INT ;
    STAT414 : INT ;
    STAT415 : INT ;
    STAT416 : WORD ;
    STAT417 : WORD ;
    STAT418 : WORD ;
    STAT419 : WORD ;
    STAT420 : WORD ;
    STAT421 : WORD ;
    STAT422 : WORD ;
    STAT423 : WORD ;
    STAT424 : WORD ;
    STAT425 : WORD ;
    STAT426 : WORD ;
    STAT427 : WORD ;
    STAT428 : WORD ;
    STAT429 : WORD ;
    STAT430 : WORD ;
    STAT431 : WORD ;
    STAT432 : WORD ;
    STAT433 : WORD ;
   END_STRUCT ;
   STAT434 : STRUCT
    STAT435 : INT ;
    STAT436 : INT ;
    STAT437 : INT ;
    STAT438 : INT ;
    STAT439 : WORD ;
    STAT440 : WORD ;
    STAT441 : INT ;
    STAT442 : INT ;
    STAT443 : INT ;
    STAT444 : INT ;
    STAT445 : INT ;
    STAT446 : INT ;
    STAT447 : WORD ;
    STAT448 : WORD ;
    STAT449 : WORD ;
    STAT450 : WORD ;
    STAT451 : WORD ;
    STAT452 : WORD ;
    STAT453 : WORD ;
    STAT454 : WORD ;
    STAT455 : WORD ;
    STAT456 : WORD ;
    STAT457 : WORD ;
    STAT458 : WORD ;
    STAT459 : WORD ;
    STAT460 : WORD ;
    STAT461 : WORD ;
    STAT462 : WORD ;
    STAT463 : WORD ;
    STAT464 : WORD ;
   END_STRUCT ;
   STAT465 : STRUCT
    STAT466 : INT ;
    STAT467 : INT ;
    STAT468 : INT ;
    STAT469 : INT ;
    STAT470 : WORD ;
    STAT471 : WORD ;
    STAT472 : INT ;
    STAT473 : INT ;
    STAT474 : INT ;
    STAT475 : INT ;
    STAT476 : INT ;
    STAT477 : INT ;
    STAT478 : WORD ;
    STAT479 : WORD ;
    STAT480 : WORD ;
    STAT481 : WORD ;
    STAT482 : WORD ;
    STAT483 : WORD ;
    STAT484 : WORD ;
    STAT485 : WORD ;
    STAT486 : WORD ;
    STAT487 : WORD ;
    STAT488 : WORD ;
    STAT489 : WORD ;
    STAT490 : WORD ;
    STAT491 : WORD ;
    STAT492 : WORD ;
    STAT493 : WORD ;
    STAT494 : WORD ;
    STAT495 : WORD ;
   END_STRUCT ;
   STAT496 : WORD ;
   STAT497 : WORD ;
  END_STRUCT ;
BEGIN
   STAT0.STAT1 := 1;
   STAT0.STAT2 := 1;
   STAT0.STAT3 := 0;
   STAT0.STAT4 := 1;
   STAT0.STAT5 := W#16#2719;
   STAT0.STAT6 := W#16#87;
   STAT0.STAT7 := 0;
   STAT0.STAT8 := 0;
   STAT0.STAT9 := 0;
   STAT0.STAT10 := 0;
   STAT0.STAT11 := 11;
   STAT0.STAT12 := 3;
   STAT0.STAT13 := W#16#2719;
   STAT0.STAT14 := W#16#87;
   STAT0.STAT15 := W#16#2222;
   STAT0.STAT16 := W#16#480;
   STAT0.STAT17 := W#16#1026;
   STAT0.STAT18 := W#16#60;
   STAT0.STAT19 := W#16#0;
   STAT0.STAT20 := W#16#0;
   STAT0.STAT21 := W#16#2720;
   STAT0.STAT22 := W#16#87;
   STAT0.STAT23 := W#16#2222;
   STAT0.STAT24 := W#16#180;
   STAT0.STAT25 := W#16#5462;
   STAT0.STAT26 := W#16#60;
   STAT0.STAT27 := W#16#0;
   STAT0.STAT28 := W#16#0;
   STAT0.STAT29 := W#16#0;
   STAT0.STAT30 := W#16#0;
   STAT31.STAT32 := 1;
   STAT31.STAT33 := 1;
   STAT31.STAT34 := 1;
   STAT31.STAT35 := 1;
   STAT31.STAT36 := W#16#2716;
   STAT31.STAT37 := W#16#87;
   STAT31.STAT38 := 0;
   STAT31.STAT39 := 0;
   STAT31.STAT40 := 0;
   STAT31.STAT41 := 0;
   STAT31.STAT42 := 11;
   STAT31.STAT43 := 3;
   STAT31.STAT44 := W#16#2716;
   STAT31.STAT45 := W#16#87;
   STAT31.STAT46 := W#16#2222;
   STAT31.STAT47 := W#16#480;
   STAT31.STAT48 := W#16#1016;
   STAT31.STAT49 := W#16#60;
   STAT31.STAT50 := W#16#0;
   STAT31.STAT51 := W#16#0;
   STAT31.STAT52 := W#16#2717;
   STAT31.STAT53 := W#16#87;
   STAT31.STAT54 := W#16#A22;
   STAT31.STAT55 := W#16#1080;
   STAT31.STAT56 := W#16#5416;
   STAT31.STAT57 := W#16#40;
   STAT31.STAT58 := W#16#0;
   STAT31.STAT59 := W#16#0;
   STAT31.STAT60 := W#16#0;
   STAT31.STAT61 := W#16#0;
   STAT62.STAT63 := 1;
   STAT62.STAT64 := 1;
   STAT62.STAT65 := 0;
   STAT62.STAT66 := 0;
   STAT62.STAT67 := W#16#9515;
   STAT62.STAT68 := W#16#1;
   STAT62.STAT69 := 0;
   STAT62.STAT70 := 0;
   STAT62.STAT71 := 0;
   STAT62.STAT72 := 0;
   STAT62.STAT73 := 11;
   STAT62.STAT74 := 3;
   STAT62.STAT75 := W#16#1;
   STAT62.STAT76 := W#16#0;
   STAT62.STAT77 := W#16#4222;
   STAT62.STAT78 := W#16#8080;
   STAT62.STAT79 := W#16#1026;
   STAT62.STAT80 := W#16#0;
   STAT62.STAT81 := W#16#0;
   STAT62.STAT82 := W#16#0;
   STAT62.STAT83 := W#16#2;
   STAT62.STAT84 := W#16#0;
   STAT62.STAT85 := W#16#4222;
   STAT62.STAT86 := W#16#8080;
   STAT62.STAT87 := W#16#1026;
   STAT62.STAT88 := W#16#0;
   STAT62.STAT89 := W#16#0;
   STAT62.STAT90 := W#16#0;
   STAT62.STAT91 := W#16#0;
   STAT62.STAT92 := W#16#0;
   STAT93.STAT94 := 1;
   STAT93.STAT95 := 1;
   STAT93.STAT96 := 0;
   STAT93.STAT97 := 0;
   STAT93.STAT98 := W#16#0;
   STAT93.STAT99 := W#16#0;
   STAT93.STAT100 := 0;
   STAT93.STAT101 := 0;
   STAT93.STAT102 := 0;
   STAT93.STAT103 := 0;
   STAT93.STAT104 := 11;
   STAT93.STAT105 := 3;
   STAT93.STAT106 := W#16#7925;
   STAT93.STAT107 := W#16#13;
   STAT93.STAT108 := W#16#221;
   STAT93.STAT109 := W#16#481;
   STAT93.STAT110 := W#16#5416;
   STAT93.STAT111 := W#16#0;
   STAT93.STAT112 := W#16#0;
   STAT93.STAT113 := W#16#0;
   STAT93.STAT114 := W#16#7926;
   STAT93.STAT115 := W#16#13;
   STAT93.STAT116 := W#16#221;
   STAT93.STAT117 := W#16#481;
   STAT93.STAT118 := W#16#4415;
   STAT93.STAT119 := W#16#0;
   STAT93.STAT120 := W#16#0;
   STAT93.STAT121 := W#16#0;
   STAT93.STAT122 := W#16#0;
   STAT93.STAT123 := W#16#0;
   STAT124.STAT125 := 1;
   STAT124.STAT126 := 1;
   STAT124.STAT127 := 0;
   STAT124.STAT128 := 1;
   STAT124.STAT129 := W#16#2716;
   STAT124.STAT130 := W#16#87;
   STAT124.STAT131 := 0;
   STAT124.STAT132 := 0;
   STAT124.STAT133 := 0;
   STAT124.STAT134 := 0;
   STAT124.STAT135 := 11;
   STAT124.STAT136 := 3;
   STAT124.STAT137 := W#16#2716;
   STAT124.STAT138 := W#16#87;
   STAT124.STAT139 := W#16#2222;
   STAT124.STAT140 := W#16#480;
   STAT124.STAT141 := W#16#1016;
   STAT124.STAT142 := W#16#60;
   STAT124.STAT143 := W#16#0;
   STAT124.STAT144 := W#16#0;
   STAT124.STAT145 := W#16#2717;
   STAT124.STAT146 := W#16#87;
   STAT124.STAT147 := W#16#A22;
   STAT124.STAT148 := W#16#1080;
   STAT124.STAT149 := W#16#5416;
   STAT124.STAT150 := W#16#40;
   STAT124.STAT151 := W#16#0;
   STAT124.STAT152 := W#16#0;
   STAT124.STAT153 := W#16#0;
   STAT124.STAT154 := W#16#0;
   STAT155.STAT156 := 1;
   STAT155.STAT157 := 1;
   STAT155.STAT158 := 1;
   STAT155.STAT159 := 1;
   STAT155.STAT160 := W#16#4602;
   STAT155.STAT161 := W#16#5;
   STAT155.STAT162 := 0;
   STAT155.STAT163 := 0;
   STAT155.STAT164 := 0;
   STAT155.STAT165 := 0;
   STAT155.STAT166 := 11;
   STAT155.STAT167 := 3;
   STAT155.STAT168 := W#16#2714;
   STAT155.STAT169 := W#16#87;
   STAT155.STAT170 := W#16#2222;
   STAT155.STAT171 := W#16#180;
   STAT155.STAT172 := W#16#5416;
   STAT155.STAT173 := W#16#60;
   STAT155.STAT174 := W#16#0;
   STAT155.STAT175 := W#16#0;
   STAT155.STAT176 := W#16#2715;
   STAT155.STAT177 := W#16#87;
   STAT155.STAT178 := W#16#2222;
   STAT155.STAT179 := W#16#180;
   STAT155.STAT180 := W#16#5462;
   STAT155.STAT181 := W#16#60;
   STAT155.STAT182 := W#16#0;
   STAT155.STAT183 := W#16#0;
   STAT155.STAT184 := W#16#0;
   STAT155.STAT185 := W#16#0;
   STAT186.STAT187 := 1;
   STAT186.STAT188 := 1;
   STAT186.STAT189 := 0;
   STAT186.STAT190 := 1;
   STAT186.STAT191 := W#16#2716;
   STAT186.STAT192 := W#16#87;
   STAT186.STAT193 := 0;
   STAT186.STAT194 := 4674;
   STAT186.STAT195 := 8704;
   STAT186.STAT196 := 2134;
   STAT186.STAT197 := 11;
   STAT186.STAT198 := 3;
   STAT186.STAT199 := W#16#2716;
   STAT186.STAT200 := W#16#87;
   STAT186.STAT201 := W#16#2222;
   STAT186.STAT202 := W#16#480;
   STAT186.STAT203 := W#16#1016;
   STAT186.STAT204 := W#16#60;
   STAT186.STAT205 := W#16#0;
   STAT186.STAT206 := W#16#0;
   STAT186.STAT207 := W#16#2717;
   STAT186.STAT208 := W#16#87;
   STAT186.STAT209 := W#16#A22;
   STAT186.STAT210 := W#16#1080;
   STAT186.STAT211 := W#16#5416;
   STAT186.STAT212 := W#16#40;
   STAT186.STAT213 := W#16#0;
   STAT186.STAT214 := W#16#0;
   STAT186.STAT215 := W#16#0;
   STAT186.STAT216 := W#16#0;
   STAT217.STAT218 := 11;
   STAT217.STAT219 := 1;
   STAT217.STAT220 := 0;
   STAT217.STAT221 := 1;
   STAT217.STAT222 := W#16#2713;
   STAT217.STAT223 := W#16#87;
   STAT217.STAT224 := 0;
   STAT217.STAT225 := 4674;
   STAT217.STAT226 := 8704;
   STAT217.STAT227 := 2134;
   STAT217.STAT228 := 11;
   STAT217.STAT229 := 3;
   STAT217.STAT230 := W#16#2713;
   STAT217.STAT231 := W#16#87;
   STAT217.STAT232 := W#16#A22;
   STAT217.STAT233 := W#16#1080;
   STAT217.STAT234 := W#16#5452;
   STAT217.STAT235 := W#16#40;
   STAT217.STAT236 := W#16#0;
   STAT217.STAT237 := W#16#0;
   STAT217.STAT238 := W#16#2714;
   STAT217.STAT239 := W#16#87;
   STAT217.STAT240 := W#16#2222;
   STAT217.STAT241 := W#16#180;
   STAT217.STAT242 := W#16#5416;
   STAT217.STAT243 := W#16#60;
   STAT217.STAT244 := W#16#0;
   STAT217.STAT245 := W#16#0;
   STAT217.STAT246 := W#16#0;
   STAT217.STAT247 := W#16#0;
   STAT248.STAT249 := 1;
   STAT248.STAT250 := 1;
   STAT248.STAT251 := 1;
   STAT248.STAT252 := 1;
   STAT248.STAT253 := W#16#0;
   STAT248.STAT254 := W#16#0;
   STAT248.STAT255 := 0;
   STAT248.STAT256 := 0;
   STAT248.STAT257 := 0;
   STAT248.STAT258 := 0;
   STAT248.STAT259 := 11;
   STAT248.STAT260 := 3;
   STAT248.STAT261 := W#16#2705;
   STAT248.STAT262 := W#16#87;
   STAT248.STAT263 := W#16#A22;
   STAT248.STAT264 := W#16#1080;
   STAT248.STAT265 := W#16#1026;
   STAT248.STAT266 := W#16#40;
   STAT248.STAT267 := W#16#0;
   STAT248.STAT268 := W#16#0;
   STAT248.STAT269 := W#16#2706;
   STAT248.STAT270 := W#16#87;
   STAT248.STAT271 := W#16#2222;
   STAT248.STAT272 := W#16#480;
   STAT248.STAT273 := W#16#1026;
   STAT248.STAT274 := W#16#60;
   STAT248.STAT275 := W#16#0;
   STAT248.STAT276 := W#16#0;
   STAT248.STAT277 := W#16#0;
   STAT248.STAT278 := W#16#0;
   STAT279.STAT280 := 0;
   STAT279.STAT281 := 0;
   STAT279.STAT282 := 0;
   STAT279.STAT283 := 0;
   STAT279.STAT284 := W#16#0;
   STAT279.STAT285 := W#16#0;
   STAT279.STAT286 := 0;
   STAT279.STAT287 := 0;
   STAT279.STAT288 := 0;
   STAT279.STAT289 := 0;
   STAT279.STAT290 := 0;
   STAT279.STAT291 := 0;
   STAT279.STAT292 := W#16#0;
   STAT279.STAT293 := W#16#0;
   STAT279.STAT294 := W#16#0;
   STAT279.STAT295 := W#16#0;
   STAT279.STAT296 := W#16#0;
   STAT279.STAT297 := W#16#0;
   STAT279.STAT298 := W#16#0;
   STAT279.STAT299 := W#16#0;
   STAT279.STAT300 := W#16#0;
   STAT279.STAT301 := W#16#0;
   STAT279.STAT302 := W#16#0;
   STAT279.STAT303 := W#16#0;
   STAT279.STAT304 := W#16#0;
   STAT279.STAT305 := W#16#0;
   STAT279.STAT306 := W#16#0;
   STAT279.STAT307 := W#16#0;
   STAT279.STAT308 := W#16#0;
   STAT279.STAT309 := W#16#0;
   STAT310.STAT311 := 11;
   STAT310.STAT312 := 0;
   STAT310.STAT313 := 0;
   STAT310.STAT314 := 0;
   STAT310.STAT315 := W#16#0;
   STAT310.STAT316 := W#16#0;
   STAT310.STAT317 := 0;
   STAT310.STAT318 := 0;
   STAT310.STAT319 := 0;
   STAT310.STAT320 := 0;
   STAT310.STAT321 := 0;
   STAT310.STAT322 := 100;
   STAT310.STAT323 := W#16#1;
   STAT310.STAT324 := W#16#0;
   STAT310.STAT325 := W#16#4222;
   STAT310.STAT326 := W#16#8080;
   STAT310.STAT327 := W#16#1026;
   STAT310.STAT328 := W#16#0;
   STAT310.STAT329 := W#16#0;
   STAT310.STAT330 := W#16#0;
   STAT310.STAT331 := W#16#2;
   STAT310.STAT332 := W#16#0;
   STAT310.STAT333 := W#16#4222;
   STAT310.STAT334 := W#16#8080;
   STAT310.STAT335 := W#16#1026;
   STAT310.STAT336 := W#16#0;
   STAT310.STAT337 := W#16#0;
   STAT310.STAT338 := W#16#0;
   STAT310.STAT339 := W#16#0;
   STAT310.STAT340 := W#16#0;
   STAT341.STAT342 := 0;
   STAT341.STAT343 := 0;
   STAT341.STAT344 := 0;
   STAT341.STAT345 := 0;
   STAT341.STAT346 := W#16#0;
   STAT341.STAT347 := W#16#0;
   STAT341.STAT348 := 0;
   STAT341.STAT349 := 0;
   STAT341.STAT350 := 0;
   STAT341.STAT351 := 0;
   STAT341.STAT352 := 0;
   STAT341.STAT353 := 0;
   STAT341.STAT354 := W#16#0;
   STAT341.STAT355 := W#16#0;
   STAT341.STAT356 := W#16#0;
   STAT341.STAT357 := W#16#0;
   STAT341.STAT358 := W#16#0;
   STAT341.STAT359 := W#16#0;
   STAT341.STAT360 := W#16#0;
   STAT341.STAT361 := W#16#0;
   STAT341.STAT362 := W#16#0;
   STAT341.STAT363 := W#16#0;
   STAT341.STAT364 := W#16#0;
   STAT341.STAT365 := W#16#0;
   STAT341.STAT366 := W#16#0;
   STAT341.STAT367 := W#16#0;
   STAT341.STAT368 := W#16#0;
   STAT341.STAT369 := W#16#0;
   STAT341.STAT370 := W#16#0;
   STAT341.STAT371 := W#16#0;
   STAT372.STAT373 := 0;
   STAT372.STAT374 := 0;
   STAT372.STAT375 := 0;
   STAT372.STAT376 := 0;
   STAT372.STAT377 := W#16#0;
   STAT372.STAT378 := W#16#0;
   STAT372.STAT379 := 0;
   STAT372.STAT380 := 0;
   STAT372.STAT381 := 0;
   STAT372.STAT382 := 0;
   STAT372.STAT383 := 0;
   STAT372.STAT384 := 0;
   STAT372.STAT385 := W#16#0;
   STAT372.STAT386 := W#16#0;
   STAT372.STAT387 := W#16#0;
   STAT372.STAT388 := W#16#0;
   STAT372.STAT389 := W#16#0;
   STAT372.STAT390 := W#16#0;
   STAT372.STAT391 := W#16#0;
   STAT372.STAT392 := W#16#0;
   STAT372.STAT393 := W#16#0;
   STAT372.STAT394 := W#16#0;
   STAT372.STAT395 := W#16#0;
   STAT372.STAT396 := W#16#0;
   STAT372.STAT397 := W#16#0;
   STAT372.STAT398 := W#16#0;
   STAT372.STAT399 := W#16#0;
   STAT372.STAT400 := W#16#0;
   STAT372.STAT401 := W#16#0;
   STAT372.STAT402 := W#16#0;
   STAT403.STAT404 := 0;
   STAT403.STAT405 := 0;
   STAT403.STAT406 := 0;
   STAT403.STAT407 := 0;
   STAT403.STAT408 := W#16#0;
   STAT403.STAT409 := W#16#0;
   STAT403.STAT410 := 0;
   STAT403.STAT411 := 0;
   STAT403.STAT412 := 0;
   STAT403.STAT413 := 0;
   STAT403.STAT414 := 0;
   STAT403.STAT415 := 0;
   STAT403.STAT416 := W#16#0;
   STAT403.STAT417 := W#16#0;
   STAT403.STAT418 := W#16#0;
   STAT403.STAT419 := W#16#0;
   STAT403.STAT420 := W#16#0;
   STAT403.STAT421 := W#16#0;
   STAT403.STAT422 := W#16#0;
   STAT403.STAT423 := W#16#0;
   STAT403.STAT424 := W#16#0;
   STAT403.STAT425 := W#16#0;
   STAT403.STAT426 := W#16#0;
   STAT403.STAT427 := W#16#0;
   STAT403.STAT428 := W#16#0;
   STAT403.STAT429 := W#16#0;
   STAT403.STAT430 := W#16#0;
   STAT403.STAT431 := W#16#0;
   STAT403.STAT432 := W#16#0;
   STAT403.STAT433 := W#16#0;
   STAT434.STAT435 := 0;
   STAT434.STAT436 := 0;
   STAT434.STAT437 := 0;
   STAT434.STAT438 := 0;
   STAT434.STAT439 := W#16#0;
   STAT434.STAT440 := W#16#0;
   STAT434.STAT441 := 0;
   STAT434.STAT442 := 0;
   STAT434.STAT443 := 0;
   STAT434.STAT444 := 0;
   STAT434.STAT445 := 0;
   STAT434.STAT446 := 0;
   STAT434.STAT447 := W#16#0;
   STAT434.STAT448 := W#16#0;
   STAT434.STAT449 := W#16#0;
   STAT434.STAT450 := W#16#0;
   STAT434.STAT451 := W#16#0;
   STAT434.STAT452 := W#16#0;
   STAT434.STAT453 := W#16#0;
   STAT434.STAT454 := W#16#0;
   STAT434.STAT455 := W#16#0;
   STAT434.STAT456 := W#16#0;
   STAT434.STAT457 := W#16#0;
   STAT434.STAT458 := W#16#0;
   STAT434.STAT459 := W#16#0;
   STAT434.STAT460 := W#16#0;
   STAT434.STAT461 := W#16#0;
   STAT434.STAT462 := W#16#0;
   STAT434.STAT463 := W#16#0;
   STAT434.STAT464 := W#16#0;
   STAT465.STAT466 := 0;
   STAT465.STAT467 := 0;
   STAT465.STAT468 := 0;
   STAT465.STAT469 := 0;
   STAT465.STAT470 := W#16#0;
   STAT465.STAT471 := W#16#0;
   STAT465.STAT472 := 0;
   STAT465.STAT473 := 0;
   STAT465.STAT474 := 0;
   STAT465.STAT475 := 0;
   STAT465.STAT476 := 0;
   STAT465.STAT477 := 0;
   STAT465.STAT478 := W#16#0;
   STAT465.STAT479 := W#16#0;
   STAT465.STAT480 := W#16#0;
   STAT465.STAT481 := W#16#0;
   STAT465.STAT482 := W#16#0;
   STAT465.STAT483 := W#16#0;
   STAT465.STAT484 := W#16#0;
   STAT465.STAT485 := W#16#0;
   STAT465.STAT486 := W#16#0;
   STAT465.STAT487 := W#16#0;
   STAT465.STAT488 := W#16#0;
   STAT465.STAT489 := W#16#0;
   STAT465.STAT490 := W#16#0;
   STAT465.STAT491 := W#16#0;
   STAT465.STAT492 := W#16#0;
   STAT465.STAT493 := W#16#0;
   STAT465.STAT494 := W#16#0;
   STAT465.STAT495 := W#16#0;
   STAT496 := W#16#0;
   STAT497 := W#16#0;
END_DATA_BLOCK

DATA_BLOCK DB 161
VERSION : 0.1


  STRUCT
   STAT0 : WORD ;
   STAT1 : WORD ;
   STAT2 : WORD ;
   STAT3 : WORD ;
   STAT4 : WORD ;
   STAT5 : WORD ;
   STAT6 : WORD ;
   STAT7 : WORD ;
   STAT8 : WORD ;
   STAT9 : WORD ;
   STAT10 : WORD ;
   STAT11 : WORD ;
   STAT12 : WORD ;
   STAT13 : WORD ;
   STAT14 : WORD ;
   STAT15 : WORD ;
   STAT16 : INT ;
   STAT17 : INT ;
   STAT18 : INT ;
   STAT19 : INT ;
   STAT20 : ARRAY  [1 .. 6 ] OF BYTE ;
   STAT21 : ARRAY  [1 .. 6 ] OF BYTE ;
   STAT22 : ARRAY  [1 .. 40 ] OF BOOL  := FALSE;
   STAT23 : ARRAY  [1 .. 40 ] OF BOOL  := FALSE;
   STAT24 : WORD ;
   STAT25 : WORD ;
   STAT26 : WORD ;
   STAT27 : WORD ;
   STAT28 : WORD ;
   STAT29 : WORD ;
   STAT30 : WORD ;
   STAT31 : ARRAY  [1 .. 7 ] OF WORD ;
   STAT32 : INT ;
   STAT33 : INT ;
   STAT34 : INT ;
   STAT35 : INT ;
   STAT36 : ARRAY  [1 .. 500 ] OF WORD ;
   STAT37 : ARRAY  [1 .. 16 ] OF BYTE ;
   STAT38 : ARRAY  [1 .. 4 ] OF BYTE ;
   STAT39 : ARRAY  [1 .. 16 ] OF BYTE ;
  END_STRUCT ;
BEGIN
   STAT0 := W#16#2720;
   STAT1 := W#16#87;
   STAT2 := W#16#2222;
   STAT3 := W#16#180;
   STAT4 := W#16#5462;
   STAT5 := W#16#60;
   STAT6 := W#16#0;
   STAT7 := W#16#0;
   STAT8 := W#16#0;
   STAT9 := W#16#0;
   STAT10 := W#16#0;
   STAT11 := W#16#0;
   STAT12 := W#16#0;
   STAT13 := W#16#0;
   STAT14 := W#16#0;
   STAT15 := W#16#0;
   STAT16 := 0;
   STAT17 := 3;
   STAT18 := 3;
   STAT19 := 0;
   STAT20[1] := B#16#14;
   STAT20[2] := B#16#1;
   STAT20[3] := B#16#0;
   STAT20[4] := B#16#0;
   STAT20[5] := B#16#94;
   STAT20[6] := B#16#2;
   STAT21[1] := B#16#0;
   STAT21[2] := B#16#0;
   STAT21[3] := B#16#0;
   STAT21[4] := B#16#0;
   STAT21[5] := B#16#0;
   STAT21[6] := B#16#0;
   STAT22[1] := FALSE;
   STAT22[2] := FALSE;
   STAT22[3] := TRUE;
   STAT22[4] := FALSE;
   STAT22[5] := FALSE;
   STAT22[6] := FALSE;
   STAT22[7] := FALSE;
   STAT22[8] := TRUE;
   STAT22[9] := FALSE;
   STAT22[10] := FALSE;
   STAT22[11] := FALSE;
   STAT22[12] := FALSE;
   STAT22[13] := FALSE;
   STAT22[14] := FALSE;
   STAT22[15] := FALSE;
   STAT22[16] := FALSE;
   STAT22[17] := FALSE;
   STAT22[18] := FALSE;
   STAT22[19] := FALSE;
   STAT22[20] := FALSE;
   STAT22[21] := FALSE;
   STAT22[22] := FALSE;
   STAT22[23] := FALSE;
   STAT22[24] := FALSE;
   STAT22[25] := FALSE;
   STAT22[26] := FALSE;
   STAT22[27] := FALSE;
   STAT22[28] := FALSE;
   STAT22[29] := FALSE;
   STAT22[30] := FALSE;
   STAT22[31] := FALSE;
   STAT22[32] := FALSE;
   STAT22[33] := FALSE;
   STAT22[34] := FALSE;
   STAT22[35] := FALSE;
   STAT22[36] := FALSE;
   STAT22[37] := FALSE;
   STAT22[38] := FALSE;
   STAT22[39] := FALSE;
   STAT22[40] := FALSE;
   STAT23[1] := FALSE;
   STAT23[2] := FALSE;
   STAT23[3] := FALSE;
   STAT23[4] := FALSE;
   STAT23[5] := FALSE;
   STAT23[6] := TRUE;
   STAT23[7] := FALSE;
   STAT23[8] := FALSE;
   STAT23[9] := FALSE;
   STAT23[10] := FALSE;
   STAT23[11] := FALSE;
   STAT23[12] := FALSE;
   STAT23[13] := FALSE;
   STAT23[14] := FALSE;
   STAT23[15] := FALSE;
   STAT23[16] := FALSE;
   STAT23[17] := FALSE;
   STAT23[18] := FALSE;
   STAT23[19] := FALSE;
   STAT23[20] := FALSE;
   STAT23[21] := FALSE;
   STAT23[22] := FALSE;
   STAT23[23] := FALSE;
   STAT23[24] := FALSE;
   STAT23[25] := FALSE;
   STAT23[26] := FALSE;
   STAT23[27] := FALSE;
   STAT23[28] := FALSE;
   STAT23[29] := FALSE;
   STAT23[30] := FALSE;
   STAT23[31] := FALSE;
   STAT23[32] := FALSE;
   STAT23[33] := FALSE;
   STAT23[34] := FALSE;
   STAT23[35] := FALSE;
   STAT23[36] := FALSE;
   STAT23[37] := FALSE;
   STAT23[38] := FALSE;
   STAT23[39] := FALSE;
   STAT23[40] := FALSE;
   STAT24 := W#16#0;
   STAT25 := W#16#0;
   STAT26 := W#16#0;
   STAT27 := W#16#0;
   STAT28 := W#16#0;
   STAT29 := W#16#0;
   STAT30 := W#16#0;
   STAT31[1] := W#16#0;
   STAT31[2] := W#16#0;
   STAT31[3] := W#16#0;
   STAT31[4] := W#16#0;
   STAT31[5] := W#16#0;
   STAT31[6] := W#16#0;
   STAT31[7] := W#16#0;
   STAT32 := 100;
   STAT33 := 90;
   STAT34 := 80;
   STAT35 := 0;
   STAT36[1] := W#16#300;
   STAT36[2] := W#16#1418;
   STAT36[3] := W#16#2435;
   STAT36[4] := W#16#B;
   STAT36[5] := W#16#2719;
   STAT36[6] := W#16#200;
   STAT36[7] := W#16#1418;
   STAT36[8] := W#16#2434;
   STAT36[9] := W#16#1;
   STAT36[10] := W#16#2718;
   STAT36[11] := W#16#500;
   STAT36[12] := W#16#1418;
   STAT36[13] := W#16#2433;
   STAT36[14] := W#16#0;
   STAT36[15] := W#16#0;
   STAT36[16] := W#16#400;
   STAT36[17] := W#16#1418;
   STAT36[18] := W#16#2432;
   STAT36[19] := W#16#0;
   STAT36[20] := W#16#0;
   STAT36[21] := W#16#300;
   STAT36[22] := W#16#1418;
   STAT36[23] := W#16#2313;
   STAT36[24] := W#16#B;
   STAT36[25] := W#16#2718;
   STAT36[26] := W#16#200;
   STAT36[27] := W#16#1418;
   STAT36[28] := W#16#2312;
   STAT36[29] := W#16#1;
   STAT36[30] := W#16#2717;
   STAT36[31] := W#16#500;
   STAT36[32] := W#16#1418;
   STAT36[33] := W#16#2312;
   STAT36[34] := W#16#0;
   STAT36[35] := W#16#0;
   STAT36[36] := W#16#400;
   STAT36[37] := W#16#1418;
   STAT36[38] := W#16#2311;
   STAT36[39] := W#16#0;
   STAT36[40] := W#16#0;
   STAT36[41] := W#16#300;
   STAT36[42] := W#16#1418;
   STAT36[43] := W#16#2208;
   STAT36[44] := W#16#B;
   STAT36[45] := W#16#2717;
   STAT36[46] := W#16#200;
   STAT36[47] := W#16#1418;
   STAT36[48] := W#16#2207;
   STAT36[49] := W#16#1;
   STAT36[50] := W#16#2716;
   STAT36[51] := W#16#500;
   STAT36[52] := W#16#1418;
   STAT36[53] := W#16#2207;
   STAT36[54] := W#16#0;
   STAT36[55] := W#16#0;
   STAT36[56] := W#16#400;
   STAT36[57] := W#16#1418;
   STAT36[58] := W#16#2206;
   STAT36[59] := W#16#0;
   STAT36[60] := W#16#0;
   STAT36[61] := W#16#300;
   STAT36[62] := W#16#1418;
   STAT36[63] := W#16#2053;
   STAT36[64] := W#16#B;
   STAT36[65] := W#16#2716;
   STAT36[66] := W#16#200;
   STAT36[67] := W#16#1418;
   STAT36[68] := W#16#2052;
   STAT36[69] := W#16#1;
   STAT36[70] := W#16#2715;
   STAT36[71] := W#16#500;
   STAT36[72] := W#16#1418;
   STAT36[73] := W#16#2052;
   STAT36[74] := W#16#0;
   STAT36[75] := W#16#0;
   STAT36[76] := W#16#400;
   STAT36[77] := W#16#1418;
   STAT36[78] := W#16#2051;
   STAT36[79] := W#16#0;
   STAT36[80] := W#16#0;
   STAT36[81] := W#16#300;
   STAT36[82] := W#16#1418;
   STAT36[83] := W#16#1933;
   STAT36[84] := W#16#B;
   STAT36[85] := W#16#2715;
   STAT36[86] := W#16#200;
   STAT36[87] := W#16#1418;
   STAT36[88] := W#16#1932;
   STAT36[89] := W#16#1;
   STAT36[90] := W#16#2714;
   STAT36[91] := W#16#500;
   STAT36[92] := W#16#1418;
   STAT36[93] := W#16#1932;
   STAT36[94] := W#16#0;
   STAT36[95] := W#16#0;
   STAT36[96] := W#16#400;
   STAT36[97] := W#16#1418;
   STAT36[98] := W#16#1931;
   STAT36[99] := W#16#0;
   STAT36[100] := W#16#0;
   STAT36[101] := W#16#300;
   STAT36[102] := W#16#1418;
   STAT36[103] := W#16#1828;
   STAT36[104] := W#16#B;
   STAT36[105] := W#16#2714;
   STAT36[106] := W#16#200;
   STAT36[107] := W#16#1418;
   STAT36[108] := W#16#1827;
   STAT36[109] := W#16#1;
   STAT36[110] := W#16#2713;
   STAT36[111] := W#16#500;
   STAT36[112] := W#16#1418;
   STAT36[113] := W#16#1827;
   STAT36[114] := W#16#0;
   STAT36[115] := W#16#0;
   STAT36[116] := W#16#400;
   STAT36[117] := W#16#1418;
   STAT36[118] := W#16#1826;
   STAT36[119] := W#16#0;
   STAT36[120] := W#16#0;
   STAT36[121] := W#16#300;
   STAT36[122] := W#16#1418;
   STAT36[123] := W#16#1714;
   STAT36[124] := W#16#B;
   STAT36[125] := W#16#2713;
   STAT36[126] := W#16#200;
   STAT36[127] := W#16#1418;
   STAT36[128] := W#16#1712;
   STAT36[129] := W#16#1;
   STAT36[130] := W#16#2712;
   STAT36[131] := W#16#500;
   STAT36[132] := W#16#1418;
   STAT36[133] := W#16#1712;
   STAT36[134] := W#16#0;
   STAT36[135] := W#16#0;
   STAT36[136] := W#16#400;
   STAT36[137] := W#16#1418;
   STAT36[138] := W#16#1711;
   STAT36[139] := W#16#0;
   STAT36[140] := W#16#0;
   STAT36[141] := W#16#300;
   STAT36[142] := W#16#1418;
   STAT36[143] := W#16#1555;
   STAT36[144] := W#16#B;
   STAT36[145] := W#16#2712;
   STAT36[146] := W#16#200;
   STAT36[147] := W#16#1418;
   STAT36[148] := W#16#1553;
   STAT36[149] := W#16#1;
   STAT36[150] := W#16#2711;
   STAT36[151] := W#16#500;
   STAT36[152] := W#16#1418;
   STAT36[153] := W#16#1553;
   STAT36[154] := W#16#0;
   STAT36[155] := W#16#0;
   STAT36[156] := W#16#400;
   STAT36[157] := W#16#1418;
   STAT36[158] := W#16#1552;
   STAT36[159] := W#16#0;
   STAT36[160] := W#16#0;
   STAT36[161] := W#16#300;
   STAT36[162] := W#16#1418;
   STAT36[163] := W#16#1450;
   STAT36[164] := W#16#B;
   STAT36[165] := W#16#2711;
   STAT36[166] := W#16#200;
   STAT36[167] := W#16#1418;
   STAT36[168] := W#16#1449;
   STAT36[169] := W#16#1;
   STAT36[170] := W#16#2710;
   STAT36[171] := W#16#500;
   STAT36[172] := W#16#1418;
   STAT36[173] := W#16#1448;
   STAT36[174] := W#16#0;
   STAT36[175] := W#16#0;
   STAT36[176] := W#16#400;
   STAT36[177] := W#16#1418;
   STAT36[178] := W#16#1447;
   STAT36[179] := W#16#0;
   STAT36[180] := W#16#0;
   STAT36[181] := W#16#300;
   STAT36[182] := W#16#1418;
   STAT36[183] := W#16#1334;
   STAT36[184] := W#16#B;
   STAT36[185] := W#16#2710;
   STAT36[186] := W#16#200;
   STAT36[187] := W#16#1418;
   STAT36[188] := W#16#1333;
   STAT36[189] := W#16#1;
   STAT36[190] := W#16#2709;
   STAT36[191] := W#16#500;
   STAT36[192] := W#16#1418;
   STAT36[193] := W#16#1332;
   STAT36[194] := W#16#0;
   STAT36[195] := W#16#0;
   STAT36[196] := W#16#400;
   STAT36[197] := W#16#1418;
   STAT36[198] := W#16#1331;
   STAT36[199] := W#16#0;
   STAT36[200] := W#16#0;
   STAT36[201] := W#16#300;
   STAT36[202] := W#16#1418;
   STAT36[203] := W#16#1218;
   STAT36[204] := W#16#B;
   STAT36[205] := W#16#2709;
   STAT36[206] := W#16#200;
   STAT36[207] := W#16#1418;
   STAT36[208] := W#16#1217;
   STAT36[209] := W#16#1;
   STAT36[210] := W#16#2708;
   STAT36[211] := W#16#500;
   STAT36[212] := W#16#1418;
   STAT36[213] := W#16#1216;
   STAT36[214] := W#16#0;
   STAT36[215] := W#16#0;
   STAT36[216] := W#16#400;
   STAT36[217] := W#16#1418;
   STAT36[218] := W#16#1215;
   STAT36[219] := W#16#0;
   STAT36[220] := W#16#0;
   STAT36[221] := W#16#300;
   STAT36[222] := W#16#1418;
   STAT36[223] := W#16#1103;
   STAT36[224] := W#16#B;
   STAT36[225] := W#16#2708;
   STAT36[226] := W#16#200;
   STAT36[227] := W#16#1418;
   STAT36[228] := W#16#1101;
   STAT36[229] := W#16#1;
   STAT36[230] := W#16#2707;
   STAT36[231] := W#16#500;
   STAT36[232] := W#16#1418;
   STAT36[233] := W#16#1101;
   STAT36[234] := W#16#0;
   STAT36[235] := W#16#0;
   STAT36[236] := W#16#400;
   STAT36[237] := W#16#1418;
   STAT36[238] := W#16#1100;
   STAT36[239] := W#16#0;
   STAT36[240] := W#16#0;
   STAT36[241] := W#16#300;
   STAT36[242] := W#16#1418;
   STAT36[243] := W#16#940;
   STAT36[244] := W#16#B;
   STAT36[245] := W#16#2707;
   STAT36[246] := W#16#200;
   STAT36[247] := W#16#1418;
   STAT36[248] := W#16#938;
   STAT36[249] := W#16#1;
   STAT36[250] := W#16#2706;
   STAT36[251] := W#16#500;
   STAT36[252] := W#16#1418;
   STAT36[253] := W#16#938;
   STAT36[254] := W#16#0;
   STAT36[255] := W#16#0;
   STAT36[256] := W#16#400;
   STAT36[257] := W#16#1418;
   STAT36[258] := W#16#937;
   STAT36[259] := W#16#0;
   STAT36[260] := W#16#0;
   STAT36[261] := W#16#300;
   STAT36[262] := W#16#1418;
   STAT36[263] := W#16#825;
   STAT36[264] := W#16#B;
   STAT36[265] := W#16#2706;
   STAT36[266] := W#16#200;
   STAT36[267] := W#16#1418;
   STAT36[268] := W#16#824;
   STAT36[269] := W#16#1;
   STAT36[270] := W#16#2705;
   STAT36[271] := W#16#500;
   STAT36[272] := W#16#1418;
   STAT36[273] := W#16#823;
   STAT36[274] := W#16#0;
   STAT36[275] := W#16#0;
   STAT36[276] := W#16#400;
   STAT36[277] := W#16#1418;
   STAT36[278] := W#16#822;
   STAT36[279] := W#16#0;
   STAT36[280] := W#16#0;
   STAT36[281] := W#16#300;
   STAT36[282] := W#16#1418;
   STAT36[283] := W#16#430;
   STAT36[284] := W#16#B;
   STAT36[285] := W#16#2705;
   STAT36[286] := W#16#200;
   STAT36[287] := W#16#1418;
   STAT36[288] := W#16#428;
   STAT36[289] := W#16#1;
   STAT36[290] := W#16#2704;
   STAT36[291] := W#16#500;
   STAT36[292] := W#16#1418;
   STAT36[293] := W#16#428;
   STAT36[294] := W#16#0;
   STAT36[295] := W#16#0;
   STAT36[296] := W#16#400;
   STAT36[297] := W#16#1418;
   STAT36[298] := W#16#427;
   STAT36[299] := W#16#0;
   STAT36[300] := W#16#0;
   STAT36[301] := W#16#300;
   STAT36[302] := W#16#1418;
   STAT36[303] := W#16#314;
   STAT36[304] := W#16#B;
   STAT36[305] := W#16#2704;
   STAT36[306] := W#16#200;
   STAT36[307] := W#16#1418;
   STAT36[308] := W#16#313;
   STAT36[309] := W#16#1;
   STAT36[310] := W#16#2703;
   STAT36[311] := W#16#500;
   STAT36[312] := W#16#1418;
   STAT36[313] := W#16#313;
   STAT36[314] := W#16#0;
   STAT36[315] := W#16#0;
   STAT36[316] := W#16#400;
   STAT36[317] := W#16#1418;
   STAT36[318] := W#16#312;
   STAT36[319] := W#16#0;
   STAT36[320] := W#16#0;
   STAT36[321] := W#16#300;
   STAT36[322] := W#16#1418;
   STAT36[323] := W#16#201;
   STAT36[324] := W#16#B;
   STAT36[325] := W#16#2703;
   STAT36[326] := W#16#200;
   STAT36[327] := W#16#1418;
   STAT36[328] := W#16#159;
   STAT36[329] := W#16#1;
   STAT36[330] := W#16#2702;
   STAT36[331] := W#16#500;
   STAT36[332] := W#16#1418;
   STAT36[333] := W#16#159;
   STAT36[334] := W#16#0;
   STAT36[335] := W#16#0;
   STAT36[336] := W#16#400;
   STAT36[337] := W#16#1418;
   STAT36[338] := W#16#158;
   STAT36[339] := W#16#0;
   STAT36[340] := W#16#0;
   STAT36[341] := W#16#300;
   STAT36[342] := W#16#1418;
   STAT36[343] := W#16#45;
   STAT36[344] := W#16#B;
   STAT36[345] := W#16#2702;
   STAT36[346] := W#16#200;
   STAT36[347] := W#16#1418;
   STAT36[348] := W#16#44;
   STAT36[349] := W#16#1;
   STAT36[350] := W#16#2701;
   STAT36[351] := W#16#500;
   STAT36[352] := W#16#1418;
   STAT36[353] := W#16#44;
   STAT36[354] := W#16#0;
   STAT36[355] := W#16#0;
   STAT36[356] := W#16#400;
   STAT36[357] := W#16#1418;
   STAT36[358] := W#16#43;
   STAT36[359] := W#16#0;
   STAT36[360] := W#16#0;
   STAT36[361] := W#16#300;
   STAT36[362] := W#16#1417;
   STAT36[363] := W#16#5924;
   STAT36[364] := W#16#B;
   STAT36[365] := W#16#2701;
   STAT36[366] := W#16#200;
   STAT36[367] := W#16#1417;
   STAT36[368] := W#16#5923;
   STAT36[369] := W#16#1;
   STAT36[370] := W#16#2700;
   STAT36[371] := W#16#500;
   STAT36[372] := W#16#1417;
   STAT36[373] := W#16#5922;
   STAT36[374] := W#16#0;
   STAT36[375] := W#16#0;
   STAT36[376] := W#16#400;
   STAT36[377] := W#16#1417;
   STAT36[378] := W#16#5921;
   STAT36[379] := W#16#0;
   STAT36[380] := W#16#0;
   STAT36[381] := W#16#300;
   STAT36[382] := W#16#1417;
   STAT36[383] := W#16#5820;
   STAT36[384] := W#16#B;
   STAT36[385] := W#16#2700;
   STAT36[386] := W#16#200;
   STAT36[387] := W#16#1417;
   STAT36[388] := W#16#5818;
   STAT36[389] := W#16#1;
   STAT36[390] := W#16#2699;
   STAT36[391] := W#16#500;
   STAT36[392] := W#16#1417;
   STAT36[393] := W#16#5818;
   STAT36[394] := W#16#0;
   STAT36[395] := W#16#0;
   STAT36[396] := W#16#400;
   STAT36[397] := W#16#1417;
   STAT36[398] := W#16#5817;
   STAT36[399] := W#16#0;
   STAT36[400] := W#16#0;
   STAT36[401] := W#16#300;
   STAT36[402] := W#16#1417;
   STAT36[403] := W#16#5707;
   STAT36[404] := W#16#B;
   STAT36[405] := W#16#2699;
   STAT36[406] := W#16#200;
   STAT36[407] := W#16#1417;
   STAT36[408] := W#16#5705;
   STAT36[409] := W#16#1;
   STAT36[410] := W#16#2698;
   STAT36[411] := W#16#500;
   STAT36[412] := W#16#1417;
   STAT36[413] := W#16#5704;
   STAT36[414] := W#16#0;
   STAT36[415] := W#16#0;
   STAT36[416] := W#16#400;
   STAT36[417] := W#16#1417;
   STAT36[418] := W#16#5703;
   STAT36[419] := W#16#0;
   STAT36[420] := W#16#0;
   STAT36[421] := W#16#300;
   STAT36[422] := W#16#1417;
   STAT36[423] := W#16#5553;
   STAT36[424] := W#16#B;
   STAT36[425] := W#16#2698;
   STAT36[426] := W#16#200;
   STAT36[427] := W#16#1417;
   STAT36[428] := W#16#5551;
   STAT36[429] := W#16#1;
   STAT36[430] := W#16#2697;
   STAT36[431] := W#16#500;
   STAT36[432] := W#16#1417;
   STAT36[433] := W#16#5551;
   STAT36[434] := W#16#0;
   STAT36[435] := W#16#0;
   STAT36[436] := W#16#400;
   STAT36[437] := W#16#1417;
   STAT36[438] := W#16#5550;
   STAT36[439] := W#16#0;
   STAT36[440] := W#16#0;
   STAT36[441] := W#16#300;
   STAT36[442] := W#16#1417;
   STAT36[443] := W#16#5439;
   STAT36[444] := W#16#B;
   STAT36[445] := W#16#2697;
   STAT36[446] := W#16#200;
   STAT36[447] := W#16#1417;
   STAT36[448] := W#16#5438;
   STAT36[449] := W#16#1;
   STAT36[450] := W#16#2696;
   STAT36[451] := W#16#500;
   STAT36[452] := W#16#1417;
   STAT36[453] := W#16#5437;
   STAT36[454] := W#16#0;
   STAT36[455] := W#16#0;
   STAT36[456] := W#16#400;
   STAT36[457] := W#16#1417;
   STAT36[458] := W#16#5436;
   STAT36[459] := W#16#0;
   STAT36[460] := W#16#0;
   STAT36[461] := W#16#300;
   STAT36[462] := W#16#1417;
   STAT36[463] := W#16#5323;
   STAT36[464] := W#16#B;
   STAT36[465] := W#16#2696;
   STAT36[466] := W#16#200;
   STAT36[467] := W#16#1417;
   STAT36[468] := W#16#5322;
   STAT36[469] := W#16#1;
   STAT36[470] := W#16#2695;
   STAT36[471] := W#16#500;
   STAT36[472] := W#16#1417;
   STAT36[473] := W#16#5321;
   STAT36[474] := W#16#0;
   STAT36[475] := W#16#0;
   STAT36[476] := W#16#400;
   STAT36[477] := W#16#1417;
   STAT36[478] := W#16#5320;
   STAT36[479] := W#16#0;
   STAT36[480] := W#16#0;
   STAT36[481] := W#16#300;
   STAT36[482] := W#16#1417;
   STAT36[483] := W#16#5208;
   STAT36[484] := W#16#B;
   STAT36[485] := W#16#2695;
   STAT36[486] := W#16#200;
   STAT36[487] := W#16#1417;
   STAT36[488] := W#16#5207;
   STAT36[489] := W#16#1;
   STAT36[490] := W#16#2694;
   STAT36[491] := W#16#500;
   STAT36[492] := W#16#1417;
   STAT36[493] := W#16#5206;
   STAT36[494] := W#16#0;
   STAT36[495] := W#16#0;
   STAT36[496] := W#16#400;
   STAT36[497] := W#16#1417;
   STAT36[498] := W#16#5205;
   STAT36[499] := W#16#0;
   STAT36[500] := W#16#0;
   STAT37[1] := B#16#0;
   STAT37[2] := B#16#87;
   STAT37[3] := B#16#27;
   STAT37[4] := B#16#19;
   STAT37[5] := B#16#22;
   STAT37[6] := B#16#22;
   STAT37[7] := B#16#80;
   STAT37[8] := B#16#4;
   STAT37[9] := B#16#26;
   STAT37[10] := B#16#10;
   STAT37[11] := B#16#60;
   STAT37[12] := B#16#0;
   STAT37[13] := B#16#0;
   STAT37[14] := B#16#0;
   STAT37[15] := B#16#0;
   STAT37[16] := B#16#0;
   STAT38[1] := B#16#0;
   STAT38[2] := B#16#0;
   STAT38[3] := B#16#0;
   STAT38[4] := B#16#0;
   STAT39[1] := B#16#0;
   STAT39[2] := B#16#0;
   STAT39[3] := B#16#0;
   STAT39[4] := B#16#0;
   STAT39[5] := B#16#0;
   STAT39[6] := B#16#0;
   STAT39[7] := B#16#0;
   STAT39[8] := B#16#0;
   STAT39[9] := B#16#0;
   STAT39[10] := B#16#0;
   STAT39[11] := B#16#0;
   STAT39[12] := B#16#0;
   STAT39[13] := B#16#0;
   STAT39[14] := B#16#0;
   STAT39[15] := B#16#0;
   STAT39[16] := B#16#0;
END_DATA_BLOCK

DATA_BLOCK DB 162
VERSION : 0.1


  STRUCT
   STAT0 : WORD ;
   STAT1 : WORD ;
   STAT2 : WORD ;
   STAT3 : WORD ;
   STAT4 : WORD ;
   STAT5 : WORD ;
   STAT6 : WORD ;
   STAT7 : WORD ;
   STAT8 : WORD ;
   STAT9 : WORD ;
   STAT10 : WORD ;
   STAT11 : WORD ;
   STAT12 : WORD ;
   STAT13 : WORD ;
   STAT14 : WORD ;
   STAT15 : WORD ;
   STAT16 : INT ;
   STAT17 : INT ;
   STAT18 : INT ;
   STAT19 : INT ;
   STAT20 : ARRAY  [1 .. 6 ] OF BYTE ;
   STAT21 : ARRAY  [1 .. 6 ] OF BYTE ;
   STAT22 : ARRAY  [1 .. 40 ] OF BOOL  := FALSE;
   STAT23 : ARRAY  [1 .. 40 ] OF BOOL  := FALSE;
   STAT24 : WORD ;
   STAT25 : WORD ;
   STAT26 : WORD ;
   STAT27 : WORD ;
   STAT28 : WORD ;
   STAT29 : WORD ;
   STAT30 : WORD ;
   STAT31 : ARRAY  [1 .. 7 ] OF WORD ;
   STAT32 : INT ;
   STAT33 : INT ;
   STAT34 : INT ;
   STAT35 : INT ;
   STAT36 : ARRAY  [1 .. 500 ] OF WORD ;
   STAT37 : ARRAY  [1 .. 16 ] OF BYTE ;
   STAT38 : ARRAY  [1 .. 4 ] OF BYTE ;
   STAT39 : ARRAY  [1 .. 16 ] OF BYTE ;
  END_STRUCT ;
BEGIN
   STAT0 := W#16#2717;
   STAT1 := W#16#87;
   STAT2 := W#16#A22;
   STAT3 := W#16#1080;
   STAT4 := W#16#5416;
   STAT5 := W#16#40;
   STAT6 := W#16#0;
   STAT7 := W#16#0;
   STAT8 := W#16#0;
   STAT9 := W#16#0;
   STAT10 := W#16#0;
   STAT11 := W#16#0;
   STAT12 := W#16#0;
   STAT13 := W#16#0;
   STAT14 := W#16#0;
   STAT15 := W#16#0;
   STAT16 := 0;
   STAT17 := 4;
   STAT18 := 3;
   STAT19 := 0;
   STAT20[1] := B#16#0;
   STAT20[2] := B#16#0;
   STAT20[3] := B#16#0;
   STAT20[4] := B#16#0;
   STAT20[5] := B#16#0;
   STAT20[6] := B#16#0;
   STAT21[1] := B#16#0;
   STAT21[2] := B#16#0;
   STAT21[3] := B#16#0;
   STAT21[4] := B#16#0;
   STAT21[5] := B#16#0;
   STAT21[6] := B#16#0;
   STAT22[1] := FALSE;
   STAT22[2] := FALSE;
   STAT22[3] := TRUE;
   STAT22[4] := FALSE;
   STAT22[5] := FALSE;
   STAT22[6] := FALSE;
   STAT22[7] := FALSE;
   STAT22[8] := TRUE;
   STAT22[9] := FALSE;
   STAT22[10] := FALSE;
   STAT22[11] := FALSE;
   STAT22[12] := FALSE;
   STAT22[13] := FALSE;
   STAT22[14] := FALSE;
   STAT22[15] := FALSE;
   STAT22[16] := FALSE;
   STAT22[17] := FALSE;
   STAT22[18] := FALSE;
   STAT22[19] := FALSE;
   STAT22[20] := FALSE;
   STAT22[21] := FALSE;
   STAT22[22] := FALSE;
   STAT22[23] := FALSE;
   STAT22[24] := FALSE;
   STAT22[25] := FALSE;
   STAT22[26] := FALSE;
   STAT22[27] := FALSE;
   STAT22[28] := FALSE;
   STAT22[29] := FALSE;
   STAT22[30] := FALSE;
   STAT22[31] := FALSE;
   STAT22[32] := FALSE;
   STAT22[33] := FALSE;
   STAT22[34] := FALSE;
   STAT22[35] := FALSE;
   STAT22[36] := FALSE;
   STAT22[37] := FALSE;
   STAT22[38] := FALSE;
   STAT22[39] := FALSE;
   STAT22[40] := FALSE;
   STAT23[1] := FALSE;
   STAT23[2] := TRUE;
   STAT23[3] := TRUE;
   STAT23[4] := TRUE;
   STAT23[5] := TRUE;
   STAT23[6] := FALSE;
   STAT23[7] := FALSE;
   STAT23[8] := FALSE;
   STAT23[9] := FALSE;
   STAT23[10] := FALSE;
   STAT23[11] := FALSE;
   STAT23[12] := FALSE;
   STAT23[13] := FALSE;
   STAT23[14] := FALSE;
   STAT23[15] := FALSE;
   STAT23[16] := FALSE;
   STAT23[17] := FALSE;
   STAT23[18] := FALSE;
   STAT23[19] := FALSE;
   STAT23[20] := FALSE;
   STAT23[21] := FALSE;
   STAT23[22] := FALSE;
   STAT23[23] := FALSE;
   STAT23[24] := FALSE;
   STAT23[25] := FALSE;
   STAT23[26] := TRUE;
   STAT23[27] := FALSE;
   STAT23[28] := FALSE;
   STAT23[29] := FALSE;
   STAT23[30] := FALSE;
   STAT23[31] := FALSE;
   STAT23[32] := FALSE;
   STAT23[33] := FALSE;
   STAT23[34] := FALSE;
   STAT23[35] := FALSE;
   STAT23[36] := FALSE;
   STAT23[37] := FALSE;
   STAT23[38] := FALSE;
   STAT23[39] := FALSE;
   STAT23[40] := FALSE;
   STAT24 := W#16#800;
   STAT25 := W#16#800;
   STAT26 := W#16#0;
   STAT27 := W#16#0;
   STAT28 := W#16#0;
   STAT29 := W#16#0;
   STAT30 := W#16#0;
   STAT31[1] := W#16#0;
   STAT31[2] := W#16#0;
   STAT31[3] := W#16#0;
   STAT31[4] := W#16#0;
   STAT31[5] := W#16#0;
   STAT31[6] := W#16#0;
   STAT31[7] := W#16#0;
   STAT32 := 100;
   STAT33 := 90;
   STAT34 := 80;
   STAT35 := 0;
   STAT36[1] := W#16#400;
   STAT36[2] := W#16#1418;
   STAT36[3] := W#16#3310;
   STAT36[4] := W#16#0;
   STAT36[5] := W#16#0;
   STAT36[6] := W#16#300;
   STAT36[7] := W#16#1418;
   STAT36[8] := W#16#2434;
   STAT36[9] := W#16#B;
   STAT36[10] := W#16#2716;
   STAT36[11] := W#16#200;
   STAT36[12] := W#16#1418;
   STAT36[13] := W#16#2432;
   STAT36[14] := W#16#1;
   STAT36[15] := W#16#2715;
   STAT36[16] := W#16#500;
   STAT36[17] := W#16#1418;
   STAT36[18] := W#16#2430;
   STAT36[19] := W#16#0;
   STAT36[20] := W#16#0;
   STAT36[21] := W#16#400;
   STAT36[22] := W#16#1418;
   STAT36[23] := W#16#2426;
   STAT36[24] := W#16#0;
   STAT36[25] := W#16#0;
   STAT36[26] := W#16#300;
   STAT36[27] := W#16#1418;
   STAT36[28] := W#16#2313;
   STAT36[29] := W#16#B;
   STAT36[30] := W#16#2715;
   STAT36[31] := W#16#200;
   STAT36[32] := W#16#1418;
   STAT36[33] := W#16#2311;
   STAT36[34] := W#16#1;
   STAT36[35] := W#16#2714;
   STAT36[36] := W#16#500;
   STAT36[37] := W#16#1418;
   STAT36[38] := W#16#2309;
   STAT36[39] := W#16#0;
   STAT36[40] := W#16#0;
   STAT36[41] := W#16#400;
   STAT36[42] := W#16#1418;
   STAT36[43] := W#16#2305;
   STAT36[44] := W#16#0;
   STAT36[45] := W#16#2714;
   STAT36[46] := W#16#300;
   STAT36[47] := W#16#1418;
   STAT36[48] := W#16#2208;
   STAT36[49] := W#16#B;
   STAT36[50] := W#16#2714;
   STAT36[51] := W#16#200;
   STAT36[52] := W#16#1418;
   STAT36[53] := W#16#2207;
   STAT36[54] := W#16#1;
   STAT36[55] := W#16#2713;
   STAT36[56] := W#16#500;
   STAT36[57] := W#16#1418;
   STAT36[58] := W#16#2204;
   STAT36[59] := W#16#0;
   STAT36[60] := W#16#0;
   STAT36[61] := W#16#400;
   STAT36[62] := W#16#1418;
   STAT36[63] := W#16#2200;
   STAT36[64] := W#16#0;
   STAT36[65] := W#16#0;
   STAT36[66] := W#16#300;
   STAT36[67] := W#16#1418;
   STAT36[68] := W#16#2106;
   STAT36[69] := W#16#B;
   STAT36[70] := W#16#2713;
   STAT36[71] := W#16#200;
   STAT36[72] := W#16#1418;
   STAT36[73] := W#16#2105;
   STAT36[74] := W#16#1;
   STAT36[75] := W#16#2712;
   STAT36[76] := W#16#500;
   STAT36[77] := W#16#1418;
   STAT36[78] := W#16#2102;
   STAT36[79] := W#16#0;
   STAT36[80] := W#16#0;
   STAT36[81] := W#16#400;
   STAT36[82] := W#16#1418;
   STAT36[83] := W#16#2044;
   STAT36[84] := W#16#0;
   STAT36[85] := W#16#0;
   STAT36[86] := W#16#300;
   STAT36[87] := W#16#1418;
   STAT36[88] := W#16#1933;
   STAT36[89] := W#16#B;
   STAT36[90] := W#16#2712;
   STAT36[91] := W#16#200;
   STAT36[92] := W#16#1418;
   STAT36[93] := W#16#1932;
   STAT36[94] := W#16#1;
   STAT36[95] := W#16#2711;
   STAT36[96] := W#16#500;
   STAT36[97] := W#16#1418;
   STAT36[98] := W#16#1929;
   STAT36[99] := W#16#0;
   STAT36[100] := W#16#0;
   STAT36[101] := W#16#400;
   STAT36[102] := W#16#1418;
   STAT36[103] := W#16#1925;
   STAT36[104] := W#16#0;
   STAT36[105] := W#16#0;
   STAT36[106] := W#16#300;
   STAT36[107] := W#16#1418;
   STAT36[108] := W#16#1827;
   STAT36[109] := W#16#B;
   STAT36[110] := W#16#2711;
   STAT36[111] := W#16#200;
   STAT36[112] := W#16#1418;
   STAT36[113] := W#16#1826;
   STAT36[114] := W#16#1;
   STAT36[115] := W#16#2710;
   STAT36[116] := W#16#500;
   STAT36[117] := W#16#1418;
   STAT36[118] := W#16#1824;
   STAT36[119] := W#16#0;
   STAT36[120] := W#16#0;
   STAT36[121] := W#16#400;
   STAT36[122] := W#16#1418;
   STAT36[123] := W#16#1820;
   STAT36[124] := W#16#0;
   STAT36[125] := W#16#0;
   STAT36[126] := W#16#300;
   STAT36[127] := W#16#1418;
   STAT36[128] := W#16#1712;
   STAT36[129] := W#16#B;
   STAT36[130] := W#16#2710;
   STAT36[131] := W#16#200;
   STAT36[132] := W#16#1418;
   STAT36[133] := W#16#1711;
   STAT36[134] := W#16#1;
   STAT36[135] := W#16#2709;
   STAT36[136] := W#16#500;
   STAT36[137] := W#16#1418;
   STAT36[138] := W#16#1708;
   STAT36[139] := W#16#0;
   STAT36[140] := W#16#0;
   STAT36[141] := W#16#400;
   STAT36[142] := W#16#1418;
   STAT36[143] := W#16#1705;
   STAT36[144] := W#16#0;
   STAT36[145] := W#16#0;
   STAT36[146] := W#16#300;
   STAT36[147] := W#16#1418;
   STAT36[148] := W#16#1557;
   STAT36[149] := W#16#B;
   STAT36[150] := W#16#2709;
   STAT36[151] := W#16#200;
   STAT36[152] := W#16#1418;
   STAT36[153] := W#16#1556;
   STAT36[154] := W#16#1;
   STAT36[155] := W#16#2708;
   STAT36[156] := W#16#500;
   STAT36[157] := W#16#1418;
   STAT36[158] := W#16#1553;
   STAT36[159] := W#16#0;
   STAT36[160] := W#16#0;
   STAT36[161] := W#16#400;
   STAT36[162] := W#16#1418;
   STAT36[163] := W#16#1551;
   STAT36[164] := W#16#0;
   STAT36[165] := W#16#0;
   STAT36[166] := W#16#300;
   STAT36[167] := W#16#1418;
   STAT36[168] := W#16#1458;
   STAT36[169] := W#16#B;
   STAT36[170] := W#16#2708;
   STAT36[171] := W#16#200;
   STAT36[172] := W#16#1418;
   STAT36[173] := W#16#1457;
   STAT36[174] := W#16#1;
   STAT36[175] := W#16#2707;
   STAT36[176] := W#16#500;
   STAT36[177] := W#16#1418;
   STAT36[178] := W#16#1455;
   STAT36[179] := W#16#0;
   STAT36[180] := W#16#0;
   STAT36[181] := W#16#400;
   STAT36[182] := W#16#1418;
   STAT36[183] := W#16#1441;
   STAT36[184] := W#16#0;
   STAT36[185] := W#16#0;
   STAT36[186] := W#16#300;
   STAT36[187] := W#16#1418;
   STAT36[188] := W#16#1333;
   STAT36[189] := W#16#B;
   STAT36[190] := W#16#2707;
   STAT36[191] := W#16#200;
   STAT36[192] := W#16#1418;
   STAT36[193] := W#16#1331;
   STAT36[194] := W#16#1;
   STAT36[195] := W#16#2706;
   STAT36[196] := W#16#500;
   STAT36[197] := W#16#1418;
   STAT36[198] := W#16#1329;
   STAT36[199] := W#16#0;
   STAT36[200] := W#16#0;
   STAT36[201] := W#16#400;
   STAT36[202] := W#16#1418;
   STAT36[203] := W#16#1325;
   STAT36[204] := W#16#0;
   STAT36[205] := W#16#0;
   STAT36[206] := W#16#300;
   STAT36[207] := W#16#1418;
   STAT36[208] := W#16#1217;
   STAT36[209] := W#16#B;
   STAT36[210] := W#16#2706;
   STAT36[211] := W#16#200;
   STAT36[212] := W#16#1418;
   STAT36[213] := W#16#1216;
   STAT36[214] := W#16#1;
   STAT36[215] := W#16#2705;
   STAT36[216] := W#16#500;
   STAT36[217] := W#16#1418;
   STAT36[218] := W#16#1213;
   STAT36[219] := W#16#0;
   STAT36[220] := W#16#0;
   STAT36[221] := W#16#400;
   STAT36[222] := W#16#1418;
   STAT36[223] := W#16#1209;
   STAT36[224] := W#16#0;
   STAT36[225] := W#16#0;
   STAT36[226] := W#16#300;
   STAT36[227] := W#16#1418;
   STAT36[228] := W#16#1101;
   STAT36[229] := W#16#B;
   STAT36[230] := W#16#2705;
   STAT36[231] := W#16#200;
   STAT36[232] := W#16#1418;
   STAT36[233] := W#16#1100;
   STAT36[234] := W#16#1;
   STAT36[235] := W#16#2704;
   STAT36[236] := W#16#500;
   STAT36[237] := W#16#1418;
   STAT36[238] := W#16#1057;
   STAT36[239] := W#16#0;
   STAT36[240] := W#16#0;
   STAT36[241] := W#16#400;
   STAT36[242] := W#16#1418;
   STAT36[243] := W#16#1054;
   STAT36[244] := W#16#0;
   STAT36[245] := W#16#0;
   STAT36[246] := W#16#300;
   STAT36[247] := W#16#1418;
   STAT36[248] := W#16#938;
   STAT36[249] := W#16#B;
   STAT36[250] := W#16#2704;
   STAT36[251] := W#16#200;
   STAT36[252] := W#16#1418;
   STAT36[253] := W#16#937;
   STAT36[254] := W#16#1;
   STAT36[255] := W#16#2703;
   STAT36[256] := W#16#500;
   STAT36[257] := W#16#1418;
   STAT36[258] := W#16#934;
   STAT36[259] := W#16#0;
   STAT36[260] := W#16#0;
   STAT36[261] := W#16#400;
   STAT36[262] := W#16#1418;
   STAT36[263] := W#16#931;
   STAT36[264] := W#16#0;
   STAT36[265] := W#16#0;
   STAT36[266] := W#16#300;
   STAT36[267] := W#16#1418;
   STAT36[268] := W#16#824;
   STAT36[269] := W#16#B;
   STAT36[270] := W#16#2703;
   STAT36[271] := W#16#200;
   STAT36[272] := W#16#1418;
   STAT36[273] := W#16#822;
   STAT36[274] := W#16#1;
   STAT36[275] := W#16#2702;
   STAT36[276] := W#16#500;
   STAT36[277] := W#16#1418;
   STAT36[278] := W#16#820;
   STAT36[279] := W#16#0;
   STAT36[280] := W#16#0;
   STAT36[281] := W#16#400;
   STAT36[282] := W#16#1418;
   STAT36[283] := W#16#816;
   STAT36[284] := W#16#0;
   STAT36[285] := W#16#0;
   STAT36[286] := W#16#300;
   STAT36[287] := W#16#1418;
   STAT36[288] := W#16#429;
   STAT36[289] := W#16#B;
   STAT36[290] := W#16#2702;
   STAT36[291] := W#16#200;
   STAT36[292] := W#16#1418;
   STAT36[293] := W#16#428;
   STAT36[294] := W#16#1;
   STAT36[295] := W#16#2701;
   STAT36[296] := W#16#500;
   STAT36[297] := W#16#1418;
   STAT36[298] := W#16#425;
   STAT36[299] := W#16#0;
   STAT36[300] := W#16#0;
   STAT36[301] := W#16#400;
   STAT36[302] := W#16#1418;
   STAT36[303] := W#16#421;
   STAT36[304] := W#16#0;
   STAT36[305] := W#16#0;
   STAT36[306] := W#16#300;
   STAT36[307] := W#16#1418;
   STAT36[308] := W#16#313;
   STAT36[309] := W#16#B;
   STAT36[310] := W#16#2701;
   STAT36[311] := W#16#200;
   STAT36[312] := W#16#1418;
   STAT36[313] := W#16#312;
   STAT36[314] := W#16#1;
   STAT36[315] := W#16#2700;
   STAT36[316] := W#16#500;
   STAT36[317] := W#16#1418;
   STAT36[318] := W#16#309;
   STAT36[319] := W#16#0;
   STAT36[320] := W#16#0;
   STAT36[321] := W#16#400;
   STAT36[322] := W#16#1418;
   STAT36[323] := W#16#305;
   STAT36[324] := W#16#0;
   STAT36[325] := W#16#0;
   STAT36[326] := W#16#300;
   STAT36[327] := W#16#1418;
   STAT36[328] := W#16#200;
   STAT36[329] := W#16#B;
   STAT36[330] := W#16#2700;
   STAT36[331] := W#16#200;
   STAT36[332] := W#16#1418;
   STAT36[333] := W#16#159;
   STAT36[334] := W#16#1;
   STAT36[335] := W#16#2699;
   STAT36[336] := W#16#500;
   STAT36[337] := W#16#1418;
   STAT36[338] := W#16#156;
   STAT36[339] := W#16#0;
   STAT36[340] := W#16#0;
   STAT36[341] := W#16#400;
   STAT36[342] := W#16#1418;
   STAT36[343] := W#16#152;
   STAT36[344] := W#16#0;
   STAT36[345] := W#16#0;
   STAT36[346] := W#16#300;
   STAT36[347] := W#16#1418;
   STAT36[348] := W#16#44;
   STAT36[349] := W#16#B;
   STAT36[350] := W#16#2699;
   STAT36[351] := W#16#200;
   STAT36[352] := W#16#1418;
   STAT36[353] := W#16#43;
   STAT36[354] := W#16#1;
   STAT36[355] := W#16#2698;
   STAT36[356] := W#16#500;
   STAT36[357] := W#16#1418;
   STAT36[358] := W#16#40;
   STAT36[359] := W#16#0;
   STAT36[360] := W#16#0;
   STAT36[361] := W#16#400;
   STAT36[362] := W#16#1418;
   STAT36[363] := W#16#37;
   STAT36[364] := W#16#0;
   STAT36[365] := W#16#0;
   STAT36[366] := W#16#300;
   STAT36[367] := W#16#1417;
   STAT36[368] := W#16#5923;
   STAT36[369] := W#16#B;
   STAT36[370] := W#16#2698;
   STAT36[371] := W#16#200;
   STAT36[372] := W#16#1417;
   STAT36[373] := W#16#5922;
   STAT36[374] := W#16#1;
   STAT36[375] := W#16#2697;
   STAT36[376] := W#16#500;
   STAT36[377] := W#16#1417;
   STAT36[378] := W#16#5920;
   STAT36[379] := W#16#0;
   STAT36[380] := W#16#0;
   STAT36[381] := W#16#400;
   STAT36[382] := W#16#1417;
   STAT36[383] := W#16#5916;
   STAT36[384] := W#16#0;
   STAT36[385] := W#16#0;
   STAT36[386] := W#16#300;
   STAT36[387] := W#16#1417;
   STAT36[388] := W#16#5818;
   STAT36[389] := W#16#B;
   STAT36[390] := W#16#2697;
   STAT36[391] := W#16#200;
   STAT36[392] := W#16#1417;
   STAT36[393] := W#16#5816;
   STAT36[394] := W#16#1;
   STAT36[395] := W#16#2696;
   STAT36[396] := W#16#500;
   STAT36[397] := W#16#1417;
   STAT36[398] := W#16#5814;
   STAT36[399] := W#16#0;
   STAT36[400] := W#16#0;
   STAT36[401] := W#16#400;
   STAT36[402] := W#16#1417;
   STAT36[403] := W#16#5810;
   STAT36[404] := W#16#0;
   STAT36[405] := W#16#0;
   STAT36[406] := W#16#300;
   STAT36[407] := W#16#1417;
   STAT36[408] := W#16#5705;
   STAT36[409] := W#16#B;
   STAT36[410] := W#16#2696;
   STAT36[411] := W#16#200;
   STAT36[412] := W#16#1417;
   STAT36[413] := W#16#5703;
   STAT36[414] := W#16#1;
   STAT36[415] := W#16#2695;
   STAT36[416] := W#16#500;
   STAT36[417] := W#16#1417;
   STAT36[418] := W#16#5701;
   STAT36[419] := W#16#0;
   STAT36[420] := W#16#0;
   STAT36[421] := W#16#400;
   STAT36[422] := W#16#1417;
   STAT36[423] := W#16#5657;
   STAT36[424] := W#16#0;
   STAT36[425] := W#16#0;
   STAT36[426] := W#16#300;
   STAT36[427] := W#16#1417;
   STAT36[428] := W#16#5551;
   STAT36[429] := W#16#B;
   STAT36[430] := W#16#2695;
   STAT36[431] := W#16#200;
   STAT36[432] := W#16#1417;
   STAT36[433] := W#16#5550;
   STAT36[434] := W#16#1;
   STAT36[435] := W#16#2694;
   STAT36[436] := W#16#500;
   STAT36[437] := W#16#1417;
   STAT36[438] := W#16#5547;
   STAT36[439] := W#16#0;
   STAT36[440] := W#16#0;
   STAT36[441] := W#16#400;
   STAT36[442] := W#16#1417;
   STAT36[443] := W#16#5544;
   STAT36[444] := W#16#0;
   STAT36[445] := W#16#0;
   STAT36[446] := W#16#300;
   STAT36[447] := W#16#1417;
   STAT36[448] := W#16#5440;
   STAT36[449] := W#16#B;
   STAT36[450] := W#16#2694;
   STAT36[451] := W#16#200;
   STAT36[452] := W#16#1417;
   STAT36[453] := W#16#5438;
   STAT36[454] := W#16#1;
   STAT36[455] := W#16#2693;
   STAT36[456] := W#16#500;
   STAT36[457] := W#16#1417;
   STAT36[458] := W#16#5436;
   STAT36[459] := W#16#0;
   STAT36[460] := W#16#0;
   STAT36[461] := W#16#400;
   STAT36[462] := W#16#1417;
   STAT36[463] := W#16#5431;
   STAT36[464] := W#16#0;
   STAT36[465] := W#16#0;
   STAT36[466] := W#16#300;
   STAT36[467] := W#16#1417;
   STAT36[468] := W#16#5337;
   STAT36[469] := W#16#B;
   STAT36[470] := W#16#2693;
   STAT36[471] := W#16#200;
   STAT36[472] := W#16#1417;
   STAT36[473] := W#16#5335;
   STAT36[474] := W#16#1;
   STAT36[475] := W#16#2692;
   STAT36[476] := W#16#500;
   STAT36[477] := W#16#1417;
   STAT36[478] := W#16#5333;
   STAT36[479] := W#16#0;
   STAT36[480] := W#16#0;
   STAT36[481] := W#16#400;
   STAT36[482] := W#16#1417;
   STAT36[483] := W#16#5315;
   STAT36[484] := W#16#0;
   STAT36[485] := W#16#0;
   STAT36[486] := W#16#300;
   STAT36[487] := W#16#1417;
   STAT36[488] := W#16#5207;
   STAT36[489] := W#16#B;
   STAT36[490] := W#16#2692;
   STAT36[491] := W#16#200;
   STAT36[492] := W#16#1417;
   STAT36[493] := W#16#5205;
   STAT36[494] := W#16#1;
   STAT36[495] := W#16#2691;
   STAT36[496] := W#16#500;
   STAT36[497] := W#16#1417;
   STAT36[498] := W#16#5203;
   STAT36[499] := W#16#0;
   STAT36[500] := W#16#0;
   STAT37[1] := B#16#0;
   STAT37[2] := B#16#87;
   STAT37[3] := B#16#27;
   STAT37[4] := B#16#16;
   STAT37[5] := B#16#22;
   STAT37[6] := B#16#22;
   STAT37[7] := B#16#80;
   STAT37[8] := B#16#4;
   STAT37[9] := B#16#16;
   STAT37[10] := B#16#10;
   STAT37[11] := B#16#60;
   STAT37[12] := B#16#0;
   STAT37[13] := B#16#0;
   STAT37[14] := B#16#0;
   STAT37[15] := B#16#0;
   STAT37[16] := B#16#0;
   STAT38[1] := B#16#0;
   STAT38[2] := B#16#0;
   STAT38[3] := B#16#0;
   STAT38[4] := B#16#0;
   STAT39[1] := B#16#0;
   STAT39[2] := B#16#0;
   STAT39[3] := B#16#0;
   STAT39[4] := B#16#0;
   STAT39[5] := B#16#0;
   STAT39[6] := B#16#0;
   STAT39[7] := B#16#0;
   STAT39[8] := B#16#0;
   STAT39[9] := B#16#0;
   STAT39[10] := B#16#0;
   STAT39[11] := B#16#0;
   STAT39[12] := B#16#0;
   STAT39[13] := B#16#0;
   STAT39[14] := B#16#0;
   STAT39[15] := B#16#0;
   STAT39[16] := B#16#0;
END_DATA_BLOCK

DATA_BLOCK DB 163
VERSION : 0.1


